// TIA Portal V17 program export: 3 tag tables, 4 data types, 12 data blocks, 34 code blocks (in call order from the OBs), 34 instance data blocks

VAR_GLOBAL   // PLC tag table "Input"
   I_D1 AT %I0.0 : Bool;
   I_D2 AT %I0.1 : Bool;
   I_D3 AT %I0.2 : Bool;
   I_D4 AT %I0.3 : Bool;
   I_D5 AT %I0.4 : Bool;
   I_D6 AT %I0.5 : Bool;
   I_D7 AT %I0.6 : Bool;
   I_D8 AT %I0.7 : Bool;
   I_D9 AT %I1.0 : Bool;
   I_Start AT %I1.1 : Bool;
   I_Reset AT %I1.2 : Bool;
   I_Stop AT %I1.3 : Bool;
   I_Auto AT %I1.4 : Bool;
   I_Manual AT %I1.5 : Bool;
   I_Estop AT %I1.6 : Bool;
   I_C1 AT %I1.7 : Bool;
   I_C2 AT %I2.0 : Bool;
   I_C3 AT %I2.1 : Bool;
   I_C4 AT %I2.2 : Bool;
   I_C5 AT %I2.3 : Bool;
   I_SendLeft AT %I2.4 : Bool;
   I_SendForward AT %I2.5 : Bool;
   I_SendRight AT %I2.6 : Bool;
   I_ResetCount AT %I2.7 : Bool;
   I_Weight AT %ID30 : Real;
END_VAR

VAR_GLOBAL   // PLC tag table "Output"
   O_W AT %Q0.0 : Bool;
   O_SendLeft AT %Q0.1 : Bool;
   O_SendRight AT %Q0.2 : Bool;
   O_SendForward AT %Q0.3 : Bool;
   O_StartLight AT %Q0.4 : Bool;
   O_ResetLight AT %Q0.5 : Bool;
   O_StopLight AT %Q0.6 : Bool;
   O_ColumnRed AT %Q0.7 : Bool;
   O_ColumnGreen AT %Q1.0 : Bool;
   O_ColumnYellow AT %Q1.1 : Bool;
   O_C1_light AT %Q1.2 : Bool;
   O_C3_light AT %Q1.4 : Bool;
   O_C4_light AT %Q1.5 : Bool;
   O_C5_light AT %Q1.6 : Bool;
   O_SendLeft_light AT %Q1.7 : Bool;
   O_SendForward_light AT %Q2.0 : Bool;
   O_SendRight_light AT %Q2.1 : Bool;
   O_ResetCount_light AT %Q2.2 : Bool;
   O_AlarmSiren AT %Q2.3 : Bool;
   O_C2_light AT %Q1.3 : Bool;
   O_LeftCount AT %QD30 : DInt;
   O_ForwardCount AT %QD34 : DInt;
   O_RightCOunt AT %QD38 : DInt;
   O_Weight AT %QD42 : Real;
   O_C1 AT %QD46 : DInt;
   O_C2 AT %QD50 : DInt;
   O_C3 AT %QD54 : DInt;
   O_C4 AT %QD58 : DInt;
END_VAR

VAR_GLOBAL   // PLC tag table "Standard-Variablentabelle"
   System_Byte AT %MB1 : Byte;
   FirstScan AT %M1.0 : Bool;
   DiagStatusUpdate AT %M1.1 : Bool;
   AlwaysTRUE AT %M1.2 : Bool;
   AlwaysFALSE AT %M1.3 : Bool;
   Clock_Byte AT %MB0 : Byte;
   Clock_10Hz AT %M0.0 : Bool;
   Clock_5Hz AT %M0.1 : Bool;
   "Clock_2.5Hz" AT %M0.2 : Bool;
   Clock_2Hz AT %M0.3 : Bool;
   "Clock_1.25Hz" AT %M0.4 : Bool;
   Clock_1Hz AT %M0.5 : Bool;
   "Clock_0.625Hz" AT %M0.6 : Bool;
   "Clock_0.5Hz" AT %M0.7 : Bool;
END_VAR

TYPE "stt_Conveyor"
// stored: IsFailsafeCompliant false
   STRUCT
      C1 : Bool;
      C2 { S7_SetPoint := 'True'} : Bool;
      C3 { S7_SetPoint := 'True'} : Bool;
      C4 { S7_SetPoint := 'True'} : Bool;
      W { S7_SetPoint := 'True'} : Bool;
      Left : Bool;
      Forward : Bool;
      Right : Bool;
   END_STRUCT;
END_TYPE

TYPE "stt_LostPackageError"
// stored: IsFailsafeCompliant false
   STRUCT
      Error_1 : Bool;
      Error_2 : Bool;
      Error_3 : Bool;
      Error_4 : Bool;
      Error_5 : Bool;
      Error_6 : Bool;
   END_STRUCT;
END_TYPE

TYPE "stt_Motor"
// stored: IsFailsafeCompliant false
   STRUCT
      Run : Bool;
      LeftTurn : Bool;
      RightTurn : Bool;
      Speed : Real;
   END_STRUCT;
END_TYPE

TYPE "stt_TimeWork"
// stored: IsFailsafeCompliant false
   STRUCT
      Seconds : USInt;
      Minute : USInt;
      Hours : USInt;
      Days : UDInt;
   END_STRUCT;
END_TYPE

DATA_BLOCK "ERR_ErrorData"   // DB27
{ S7_Optimized_Access := 'TRUE' }
VERSION : 0.1
// stored: AutoNumber true, IsOnlyStoredInLoadMemory false, IsRetainMemResEnabled false, IsWriteProtectedInAS false, MemoryReserve 100
   VAR
      ErrorChangeMode : Bool;
      ErrorEmergencyStop : Bool;
      ErrorLostPackage_B { S7_SetPoint := 'True'} : Bool;
      ErrorLostPackage : "stt_LostPackageError";
   END_VAR
BEGIN
END_DATA_BLOCK

DATA_BLOCK "TST_ChooseModeData"   // DB4
{ S7_Optimized_Access := 'TRUE' }
VERSION : 0.1
// stored: AutoNumber true, IsOnlyStoredInLoadMemory false, IsRetainMemResEnabled false, IsWriteProtectedInAS false, MemoryReserve 100
   VAR
      Auto : Bool;
      Manual : Bool;
      inAuto : Bool;
      inManual : Bool;
   END_VAR
BEGIN
END_DATA_BLOCK

DATA_BLOCK "TST_ControlLineData"   // DB7
{ S7_Optimized_Access := 'TRUE' }
VERSION : 0.1
// stored: AutoNumber true, IsOnlyStoredInLoadMemory false, IsRetainMemResEnabled false, IsWriteProtectedInAS false, MemoryReserve 100
   VAR
      inAuto : Bool;
      inManual : Bool;
      inStart : Bool;
      inStop : Bool;
      inGlobalError : Bool;
      inRunLine : Bool;
      StartLine : Bool;
      StopLine : Bool;
      StartAlarmSiren : Bool;
   END_VAR
BEGIN
END_DATA_BLOCK

DATA_BLOCK "LOG_LogicData"   // DB55
{ S7_Optimized_Access := 'TRUE' }
VERSION : 0.1
// stored: AutoNumber true, IsOnlyStoredInLoadMemory false, IsRetainMemResEnabled false, IsWriteProtectedInAS false, MemoryReserve 100
   VAR
      ConveyorsManual : "stt_Conveyor";
      ConveyorsAuto : "stt_Conveyor";
   END_VAR
BEGIN
END_DATA_BLOCK

DATA_BLOCK "HW_HardwareData"   // DB16
{ S7_Optimized_Access := 'TRUE' }
VERSION : 0.1
// stored: AutoNumber true, IsOnlyStoredInLoadMemory false, IsRetainMemResEnabled false, IsWriteProtectedInAS false, MemoryReserve 100
   VAR
      C1 : "stt_Motor";
      C2 { S7_SetPoint := 'True'} : "stt_Motor";
      C3 { S7_SetPoint := 'True'} : "stt_Motor";
      C4 { S7_SetPoint := 'True'} : "stt_Motor";
      W { S7_SetPoint := 'True'} : Bool;
      SendLeft : Bool;
      SendForward : Bool;
      SendRight : Bool;
   END_VAR
BEGIN
END_DATA_BLOCK

DATA_BLOCK "LOG_ConveyorWorkTime"   // DB47
{ S7_Optimized_Access := 'TRUE' }
VERSION : 0.1
// stored: AutoNumber true, IsOnlyStoredInLoadMemory false, IsRetainMemResEnabled false, IsWriteProtectedInAS false, MemoryReserve 20
   VAR RETAIN
      T1 { S7_SetPoint := 'True'} : "stt_TimeWork";
      T2 { S7_SetPoint := 'True'} : "stt_TimeWork";
      T3 { S7_SetPoint := 'True'} : "stt_TimeWork";
   END_VAR
   VAR
      T4 { S7_SetPoint := 'True'} : "stt_TimeWork";
      W { S7_SetPoint := 'True'} : "stt_TimeWork";
      O { S7_SetPoint := 'True'} : "stt_TimeWork";
   END_VAR
BEGIN
END_DATA_BLOCK

DATA_BLOCK "LOG_LineModeTurnOn"   // DB46
{ S7_Optimized_Access := 'TRUE' }
VERSION : 0.1
// stored: AutoNumber true, IsOnlyStoredInLoadMemory false, IsRetainMemResEnabled false, IsWriteProtectedInAS false, MemoryReserve 20
   VAR RETAIN
      ModeAuto : UDInt;
      ModeManual : UDInt;
   END_VAR
   VAR
      EmergencyButton : Int;
      ErrorLostPackage : UDInt;
      ErrorChangeMode : UDInt;
   END_VAR
BEGIN
END_DATA_BLOCK

DATA_BLOCK "LOG_LineTimeStatistic"   // DB44
{ S7_Optimized_Access := 'TRUE' }
VERSION : 0.1
// stored: AutoNumber true, IsOnlyStoredInLoadMemory false, IsRetainMemResEnabled false, IsWriteProtectedInAS false, MemoryReserve 20
   VAR RETAIN
      StartLine { S7_SetPoint := 'True'} : "stt_TimeWork";
      StopLine { S7_SetPoint := 'True'} : "stt_TimeWork";
      AutoMode { S7_SetPoint := 'True'} : "stt_TimeWork";
      ManualMode { S7_SetPoint := 'True'} : "stt_TimeWork";
      Error { S7_SetPoint := 'True'} : "stt_TimeWork";
   END_VAR
BEGIN
END_DATA_BLOCK

DATA_BLOCK "LOG_StatisticData"   // DB43
{ S7_Optimized_Access := 'TRUE' }
VERSION : 0.1
// stored: AutoNumber true, IsOnlyStoredInLoadMemory false, IsRetainMemResEnabled false, IsWriteProtectedInAS false, MemoryReserve 100
   VAR
      P_StartLine : Bool;
   END_VAR
BEGIN
END_DATA_BLOCK

DATA_BLOCK "LOG_TotalProduction"   // DB39
{ S7_Optimized_Access := 'TRUE' }
VERSION : 0.1
// stored: AutoNumber true, IsOnlyStoredInLoadMemory false, IsRetainMemResEnabled false, IsWriteProtectedInAS false, MemoryReserve 100
   VAR
      SmallPackage : Int;
      MediumPackage : Int;
      LargePackage : Int;
   END_VAR
BEGIN
END_DATA_BLOCK

DATA_BLOCK "HW_WeightData"   // DB22
{ S7_Optimized_Access := 'TRUE' }
VERSION : 0.1
// stored: AutoNumber true, IsOnlyStoredInLoadMemory false, IsRetainMemResEnabled false, IsWriteProtectedInAS false, MemoryReserve 100
   VAR
      WeightFilter : Real;
      P_D2 : Bool;
      WeightOfSmallPackage : Real;
      WeightOfLargePackage : Real;
      IsSmallPackage : Bool;
      IsMediumPackage : Bool;
      IsLargePackage : Bool;
   END_VAR
BEGIN
END_DATA_BLOCK

DATA_BLOCK "MAN_LineModeData"   // DB1
{ S7_Optimized_Access := 'TRUE' }
VERSION : 0.1
// stored: AutoNumber true, IsOnlyStoredInLoadMemory false, IsRetainMemResEnabled false, IsWriteProtectedInAS false, MemoryReserve 100
   VAR
      Start : Bool;
      Stop : Bool;
      Manual : Bool;
      Auto : Bool;
      Error : Bool;
      RunLine : Bool;
      AlarmSiren : Bool;
   END_VAR
BEGIN
END_DATA_BLOCK

ORGANIZATION_BLOCK "Main"   // OB1, LAD, ProgramCycle
TITLE = "Main Program Sweep (Cycle)"
{ S7_Optimized_Access := 'TRUE' }
VERSION : 0.1
// stored: AutoNumber true, IsIECCheckEnabled false, SetENOAutomatically false
   VAR_INPUT
      Initial_Call : Bool;   // Initial call of this OB
      Remanence : Bool;   // =True, if remanent data are available
   END_VAR
BEGIN

REGION Network 1: Connection of PLC with FactoryIO
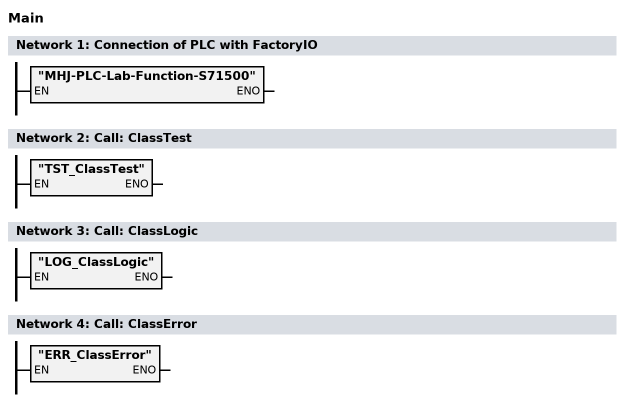
   RUNG wire#powerrail
      "MHJ-PLC-Lab-Function-S71500"()
   END_RUNG
   // the same network as SCL:
   "MHJ-PLC-Lab-Function-S71500"();
END_REGION

REGION Network 2: Call: ClassTest
   RUNG wire#powerrail
      "TST_ClassTest"()
   END_RUNG
   // the same network as SCL:
   "TST_ClassTest"();
END_REGION

REGION Network 3: Call: ClassLogic
   RUNG wire#powerrail
      "LOG_ClassLogic"()
   END_RUNG
   // the same network as SCL:
   "LOG_ClassLogic"();
END_REGION

REGION Network 4: Call: ClassError
   RUNG wire#powerrail
      "ERR_ClassError"()
   END_RUNG
   // the same network as SCL:
   "ERR_ClassError"();
END_REGION
END_ORGANIZATION_BLOCK

FUNCTION "TST_ClassTest" : Void   // FC2, LAD
{ S7_Optimized_Access := 'TRUE' }
VERSION : 0.1
// stored: AutoNumber true, IsIECCheckEnabled false, SetENOAutomatically false, UDAEnableTagReadback false
BEGIN

REGION Network 1: Call: ChooseMode
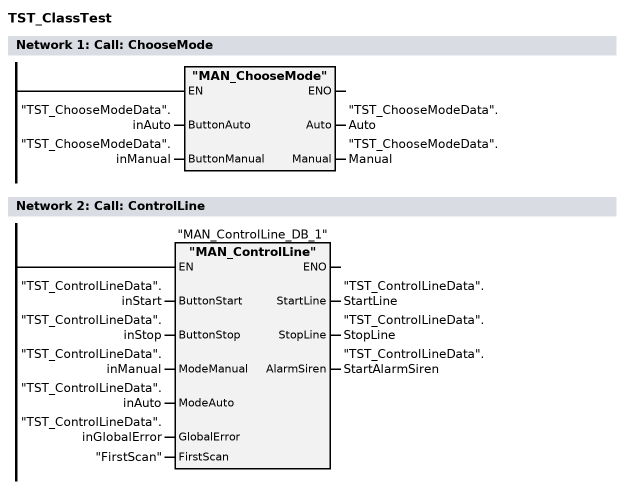
   RUNG wire#powerrail
      "MAN_ChooseMode"(ButtonAuto := "TST_ChooseModeData".inAuto, ButtonManual := "TST_ChooseModeData".inManual, Auto => "TST_ChooseModeData".Auto, Manual => "TST_ChooseModeData".Manual)
   END_RUNG
   // the same network as SCL:
   "MAN_ChooseMode"(ButtonAuto := "TST_ChooseModeData".inAuto,
                    ButtonManual := "TST_ChooseModeData".inManual,
                    Auto => "TST_ChooseModeData".Auto,
                    Manual => "TST_ChooseModeData".Manual);
END_REGION

REGION Network 2: Call: ControlLine
   RUNG wire#powerrail
      "MAN_ControlLine_DB_1"(ButtonStart := "TST_ControlLineData".inStart, ButtonStop := "TST_ControlLineData".inStop, ModeManual := "TST_ControlLineData".inManual, ModeAuto := "TST_ControlLineData".inAuto, GlobalError := "TST_ControlLineData".inGlobalError, FirstScan := "FirstScan", StartLine => "TST_ControlLineData".StartLine, StopLine => "TST_ControlLineData".StopLine, AlarmSiren => "TST_ControlLineData".StartAlarmSiren)
   END_RUNG
   // the same network as SCL:
   "MAN_ControlLine_DB_1"(ButtonStart := "TST_ControlLineData".inStart,   // "MAN_ControlLine"
                          ButtonStop := "TST_ControlLineData".inStop,
                          ModeManual := "TST_ControlLineData".inManual,
                          ModeAuto := "TST_ControlLineData".inAuto,
                          GlobalError := "TST_ControlLineData".inGlobalError,
                          FirstScan := "FirstScan",
                          StartLine => "TST_ControlLineData".StartLine,
                          StopLine => "TST_ControlLineData".StopLine,
                          AlarmSiren => "TST_ControlLineData".StartAlarmSiren);
END_REGION
END_FUNCTION

FUNCTION "MAN_ChooseMode" : Void   // FC7, LAD
{ S7_Optimized_Access := 'TRUE' }
VERSION : 0.1
// stored: AutoNumber true, IsIECCheckEnabled false, SetENOAutomatically false, UDAEnableTagReadback false
   VAR_INPUT
      ButtonAuto : Bool;
      ButtonManual : Bool;
   END_VAR
   VAR_OUTPUT
      Auto : Bool;
      Manual : Bool;
   END_VAR
BEGIN

REGION Network 1
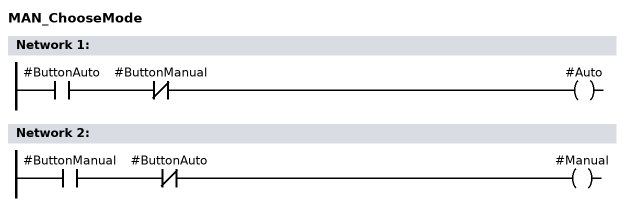
   RUNG wire#powerrail
      Contact( #ButtonAuto )
      I_Contact( #ButtonManual )
      Coil( #Auto )
   END_RUNG
   // the same network as SCL:
   #Auto := #ButtonAuto AND NOT #ButtonManual;
END_REGION

REGION Network 2
   RUNG wire#powerrail
      Contact( #ButtonManual )
      I_Contact( #ButtonAuto )
      Coil( #Manual )
   END_RUNG
   // the same network as SCL:
   #Manual := #ButtonManual AND NOT #ButtonAuto;
END_REGION
END_FUNCTION

FUNCTION_BLOCK "MAN_ControlLine"   // FB2, LAD
TITLE = Control Line - Sequential algorithm
{ S7_Optimized_Access := 'TRUE' }
VERSION : 0.1
// stored: AutoNumber true, IsIECCheckEnabled false, IsRetainMemResEnabled false, MemoryReserve 100, SetENOAutomatically false, UDAEnableTagReadback false
   VAR_INPUT
      ButtonStart : Bool;
      ButtonStop : Bool;
      ModeManual : Bool;
      ModeAuto : Bool;
      GlobalError : Bool;
      FirstScan : Bool;
   END_VAR
   VAR_OUTPUT
      StartLine : Bool;
      StopLine : Bool;
      AlarmSiren : Bool;
   END_VAR
   VAR
      s1 : Bool;
      s2 : Bool;
      s3 : Bool;
      s4 : Bool;
      P_ButtonStart_1 : Bool;
      P_ButtonStart_2 : Bool;
      IEC_Timer_0_Instance { ExternalAccessible := 'False'; ExternalVisible := 'False'; ExternalWritable := 'False'} : TP_TIME;
      Run { S7_SetPoint := 'True'} : Bool;
      N_Run : Bool;
   END_VAR
   VAR_TEMP   // added for the SCL form of the ladder/FBD networks
      _w1 : Bool;
   END_VAR
BEGIN

REGION Network 1: Step 2-1
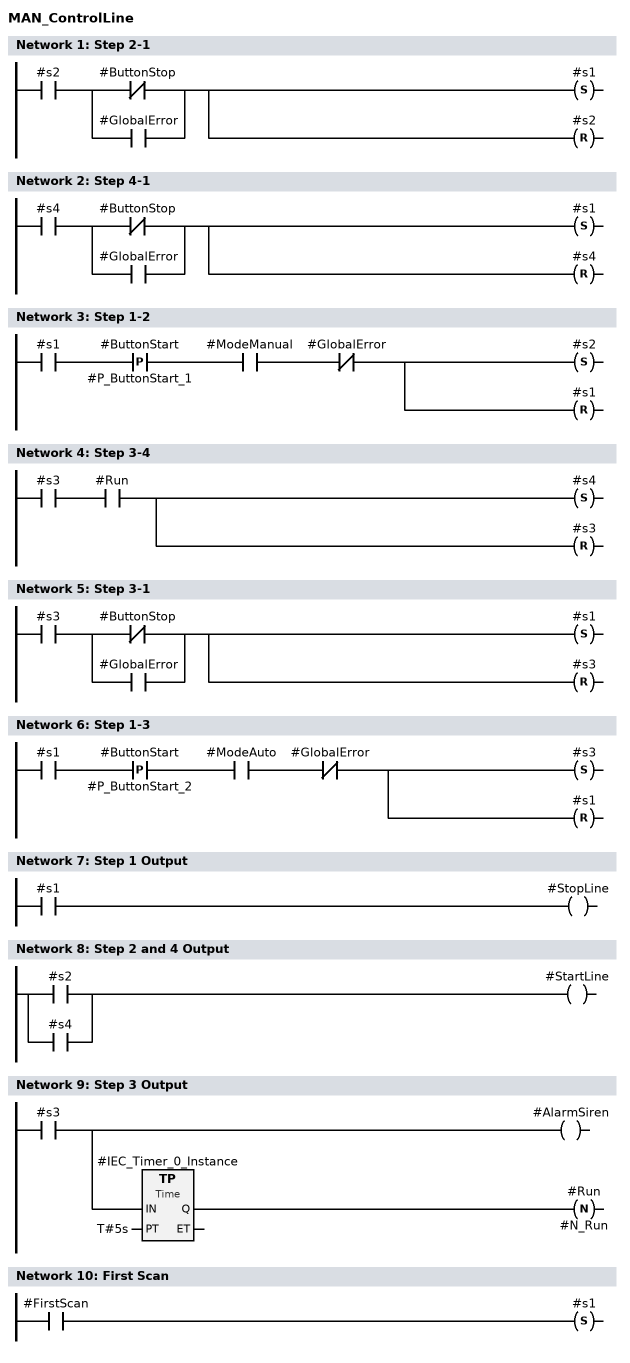
   RUNG wire#powerrail
      Contact( #s2 )
      wire#w1
      I_Contact( #ButtonStop )
      wire#w2
      S_Coil( #s1 )
   END_RUNG
   RUNG wire#w1
      Contact( #GlobalError )
   END_RUNG wire#w2
   RUNG wire#w2
      R_Coil( #s2 )
   END_RUNG
   // the same network as SCL:
   IF #s2 AND (NOT #ButtonStop OR #GlobalError) THEN
       #s1 := TRUE;
       #s2 := FALSE;
   END_IF;
END_REGION

REGION Network 2: Step 4-1
   RUNG wire#powerrail
      Contact( #s4 )
      wire#w1
      I_Contact( #ButtonStop )
      wire#w2
      S_Coil( #s1 )
   END_RUNG
   RUNG wire#w1
      Contact( #GlobalError )
   END_RUNG wire#w2
   RUNG wire#w2
      R_Coil( #s4 )
   END_RUNG
   // the same network as SCL:
   IF #s4 AND (NOT #ButtonStop OR #GlobalError) THEN
       #s1 := TRUE;
       #s4 := FALSE;
   END_IF;
END_REGION

REGION Network 3: Step 1-2
   RUNG wire#powerrail
      Contact( #s1 )
      P_Contact(operand := #ButtonStart, bit := #P_ButtonStart_1)
      Contact( #ModeManual )
      I_Contact( #GlobalError )
      wire#w1
      S_Coil( #s2 )
   END_RUNG
   RUNG wire#w1
      R_Coil( #s1 )
   END_RUNG
   // the same network as SCL:
   #_w1 := #s1 AND #ButtonStart AND NOT #P_ButtonStart_1;   // rising edge of #ButtonStart
   #P_ButtonStart_1 := #ButtonStart;
   IF #_w1 AND #ModeManual AND NOT #GlobalError THEN
       #s2 := TRUE;
       #s1 := FALSE;
   END_IF;
END_REGION

REGION Network 4: Step 3-4
   RUNG wire#powerrail
      Contact( #s3 )
      Contact( #Run )
      wire#w1
      S_Coil( #s4 )
   END_RUNG
   RUNG wire#w1
      R_Coil( #s3 )
   END_RUNG
   // the same network as SCL:
   IF #s3 AND #Run THEN
       #s4 := TRUE;
       #s3 := FALSE;
   END_IF;
END_REGION

REGION Network 5: Step 3-1
   RUNG wire#powerrail
      Contact( #s3 )
      wire#w1
      I_Contact( #ButtonStop )
      wire#w2
      S_Coil( #s1 )
   END_RUNG
   RUNG wire#w1
      Contact( #GlobalError )
   END_RUNG wire#w2
   RUNG wire#w2
      R_Coil( #s3 )
   END_RUNG
   // the same network as SCL:
   IF #s3 AND (NOT #ButtonStop OR #GlobalError) THEN
       #s1 := TRUE;
       #s3 := FALSE;
   END_IF;
END_REGION

REGION Network 6: Step 1-3
   RUNG wire#powerrail
      Contact( #s1 )
      P_Contact(operand := #ButtonStart, bit := #P_ButtonStart_2)
      Contact( #ModeAuto )
      I_Contact( #GlobalError )
      wire#w1
      S_Coil( #s3 )
   END_RUNG
   RUNG wire#w1
      R_Coil( #s1 )
   END_RUNG
   // the same network as SCL:
   #_w1 := #s1 AND #ButtonStart AND NOT #P_ButtonStart_2;   // rising edge of #ButtonStart
   #P_ButtonStart_2 := #ButtonStart;
   IF #_w1 AND #ModeAuto AND NOT #GlobalError THEN
       #s3 := TRUE;
       #s1 := FALSE;
   END_IF;
END_REGION

REGION Network 7: Step 1 Output
   RUNG wire#powerrail
      Contact( #s1 )
      Coil( #StopLine )
   END_RUNG
   // the same network as SCL:
   #StopLine := #s1;
END_REGION

REGION Network 8: Step 2 and 4 Output
   RUNG wire#powerrail
      Contact( #s2 )
      wire#w1
      Coil( #StartLine )
   END_RUNG
   RUNG wire#powerrail
      Contact( #s4 )
   END_RUNG wire#w1
   // the same network as SCL:
   #StartLine := #s2 OR #s4;
END_REGION

REGION Network 9: Step 3 Output
   #AlarmSiren := #s3;
   #IEC_Timer_0_Instance(IN := #s3, PT := T#5s);   // TP
   #Run := NOT #IEC_Timer_0_Instance.Q AND #N_Run;   // falling edge
   #N_Run := #IEC_Timer_0_Instance.Q;
END_REGION

REGION Network 10: First Scan
   RUNG wire#powerrail
      Contact( #FirstScan )
      S_Coil( #s1 )
   END_RUNG
   // the same network as SCL:
   IF #FirstScan THEN #s1 := TRUE; END_IF;
END_REGION
END_FUNCTION_BLOCK

FUNCTION "LOG_ClassLogic" : Void   // FC4, LAD
{ S7_Optimized_Access := 'TRUE' }
VERSION : 0.1
// stored: AutoNumber true, IsIECCheckEnabled false, SetENOAutomatically false, UDAEnableTagReadback false
BEGIN

REGION Network 1: Call: Mode
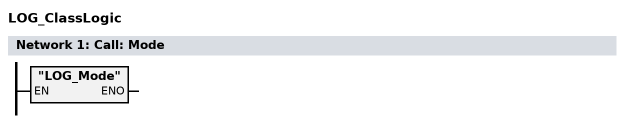
   RUNG wire#powerrail
      "LOG_Mode"()
   END_RUNG
   // the same network as SCL:
   "LOG_Mode"();
END_REGION
END_FUNCTION

FUNCTION "LOG_Mode" : Void   // FC13, LAD
{ S7_Optimized_Access := 'TRUE' }
VERSION : 0.1
// stored: AutoNumber true, IsIECCheckEnabled false, SetENOAutomatically false, UDAEnableTagReadback false
BEGIN

REGION Network 1: Call: AutoControle
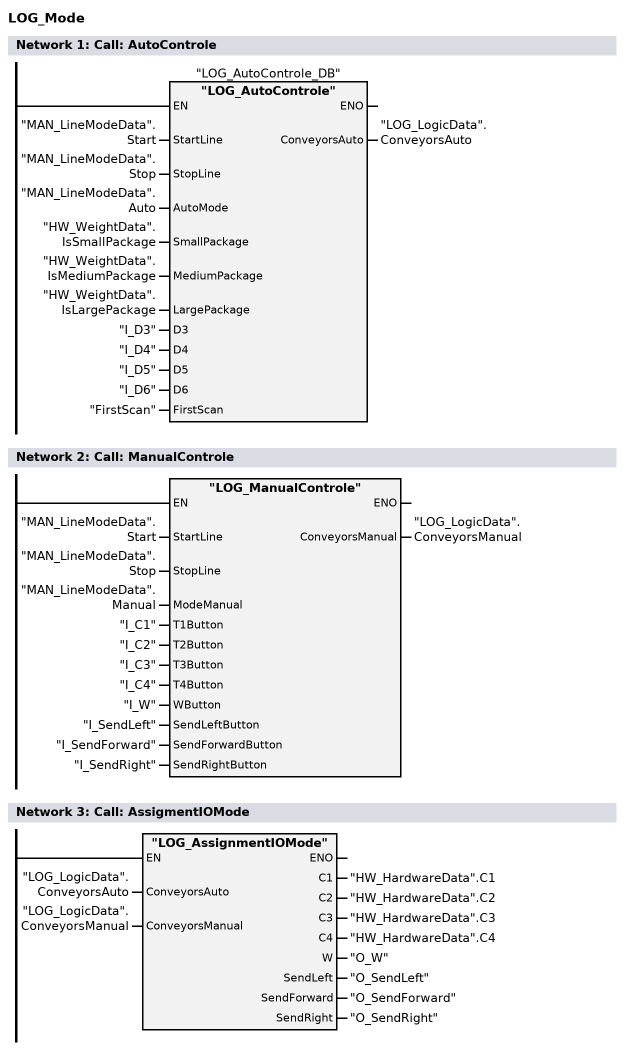
   RUNG wire#powerrail
      "LOG_AutoControle_DB"(StartLine := "MAN_LineModeData".Start, StopLine := "MAN_LineModeData".Stop, AutoMode := "MAN_LineModeData".Auto, SmallPackage := "HW_WeightData".IsSmallPackage, MediumPackage := "HW_WeightData".IsMediumPackage, LargePackage := "HW_WeightData".IsLargePackage, D3 := "I_D3", D4 := "I_D4", D5 := "I_D5", D6 := "I_D6", FirstScan := "FirstScan", ConveyorsAuto => "LOG_LogicData".ConveyorsAuto)
   END_RUNG
   // the same network as SCL:
   "LOG_AutoControle_DB"(StartLine := "MAN_LineModeData".Start,   // "LOG_AutoControle"
                         StopLine := "MAN_LineModeData".Stop,
                         AutoMode := "MAN_LineModeData".Auto,
                         SmallPackage := "HW_WeightData".IsSmallPackage,
                         MediumPackage := "HW_WeightData".IsMediumPackage,
                         LargePackage := "HW_WeightData".IsLargePackage,
                         D3 := "I_D3",
                         D4 := "I_D4",
                         D5 := "I_D5",
                         D6 := "I_D6",
                         FirstScan := "FirstScan",
                         ConveyorsAuto => "LOG_LogicData".ConveyorsAuto);
END_REGION

REGION Network 2: Call: ManualControle
   RUNG wire#powerrail
      "LOG_ManualControle"(StartLine := "MAN_LineModeData".Start, StopLine := "MAN_LineModeData".Stop, ModeManual := "MAN_LineModeData".Manual, T1Button := "I_C1", T2Button := "I_C2", T3Button := "I_C3", T4Button := "I_C4", WButton := "I_W", SendLeftButton := "I_SendLeft", SendForwardButton := "I_SendForward", SendRightButton := "I_SendRight", ConveyorsManual => "LOG_LogicData".ConveyorsManual)
   END_RUNG
   // the same network as SCL:
   "LOG_ManualControle"(StartLine := "MAN_LineModeData".Start,
                        StopLine := "MAN_LineModeData".Stop,
                        ModeManual := "MAN_LineModeData".Manual,
                        T1Button := "I_C1",
                        T2Button := "I_C2",
                        T3Button := "I_C3",
                        T4Button := "I_C4",
                        WButton := "I_W",
                        SendLeftButton := "I_SendLeft",
                        SendForwardButton := "I_SendForward",
                        SendRightButton := "I_SendRight",
                        ConveyorsManual => "LOG_LogicData".ConveyorsManual);
END_REGION

REGION Network 3: Call: AssigmentIOMode
   RUNG wire#powerrail
      "LOG_AssignmentIOMode"(ConveyorsAuto := "LOG_LogicData".ConveyorsAuto, ConveyorsManual := "LOG_LogicData".ConveyorsManual, C1 => "HW_HardwareData".C1, C2 => "HW_HardwareData".C2, C3 => "HW_HardwareData".C3, C4 => "HW_HardwareData".C4, W => "O_W", SendLeft => "O_SendLeft", SendForward => "O_SendForward", SendRight => "O_SendRight")
   END_RUNG
   // the same network as SCL:
   "LOG_AssignmentIOMode"(ConveyorsAuto := "LOG_LogicData".ConveyorsAuto,
                          ConveyorsManual := "LOG_LogicData".ConveyorsManual,
                          C1 => "HW_HardwareData".C1,
                          C2 => "HW_HardwareData".C2,
                          C3 => "HW_HardwareData".C3,
                          C4 => "HW_HardwareData".C4,
                          W => "O_W",
                          SendLeft => "O_SendLeft",
                          SendForward => "O_SendForward",
                          SendRight => "O_SendRight");
END_REGION
END_FUNCTION

FUNCTION_BLOCK "LOG_AutoControle"   // FB5, LAD
TITLE = Auto Controle - Sequential algorithm
{ S7_Optimized_Access := 'TRUE' }
VERSION : 0.1
// stored: AutoNumber true, IsIECCheckEnabled false, IsRetainMemResEnabled false, MemoryReserve 100, SetENOAutomatically false, UDAEnableTagReadback false
   VAR_INPUT
      StartLine : Bool;
      StopLine : Bool;
      AutoMode : Bool;
      SmallPackage : Bool;
      MediumPackage : Bool;
      LargePackage : Bool;
      D3 : Bool;
      D4 : Bool;
      D5 : Bool;
      D6 : Bool;
      FirstScan : Bool;
   END_VAR
   VAR_OUTPUT
      ConveyorsAuto : "stt_Conveyor";
   END_VAR
   VAR
      s1 : Bool;
      s2 : Bool;
      s3 : Bool;
      s4 : Bool;
      s5 : Bool;
      P_D3_1 : Bool;
      P_D3_2 : Bool;
      P_D3_3 : Bool;
      N_D4 : Bool;
      N_D5 : Bool;
      N_D6 : Bool;
   END_VAR
   VAR_TEMP   // added for the SCL form of the ladder/FBD networks
      _w1 : Bool;
   END_VAR
BEGIN

REGION Network 1: Step 3-2
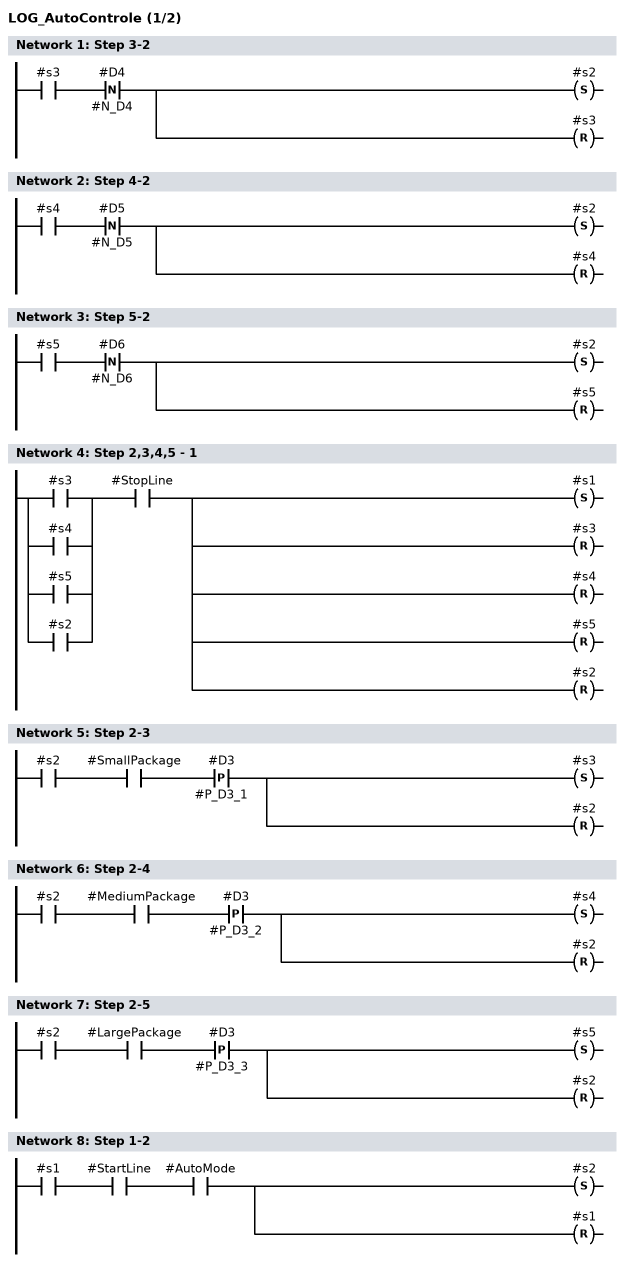
   RUNG wire#powerrail
      Contact( #s3 )
      N_Contact(operand := #D4, bit := #N_D4)
      wire#w1
      S_Coil( #s2 )
   END_RUNG
   RUNG wire#w1
      R_Coil( #s3 )
   END_RUNG
   // the same network as SCL:
   #_w1 := #s3 AND NOT #D4 AND #N_D4;   // falling edge of #D4
   #N_D4 := #D4;
   IF #_w1 THEN
       #s2 := TRUE;
       #s3 := FALSE;
   END_IF;
END_REGION

REGION Network 2: Step 4-2
   RUNG wire#powerrail
      Contact( #s4 )
      N_Contact(operand := #D5, bit := #N_D5)
      wire#w1
      S_Coil( #s2 )
   END_RUNG
   RUNG wire#w1
      R_Coil( #s4 )
   END_RUNG
   // the same network as SCL:
   #_w1 := #s4 AND NOT #D5 AND #N_D5;   // falling edge of #D5
   #N_D5 := #D5;
   IF #_w1 THEN
       #s2 := TRUE;
       #s4 := FALSE;
   END_IF;
END_REGION

REGION Network 3: Step 5-2
   RUNG wire#powerrail
      Contact( #s5 )
      N_Contact(operand := #D6, bit := #N_D6)
      wire#w1
      S_Coil( #s2 )
   END_RUNG
   RUNG wire#w1
      R_Coil( #s5 )
   END_RUNG
   // the same network as SCL:
   #_w1 := #s5 AND NOT #D6 AND #N_D6;   // falling edge of #D6
   #N_D6 := #D6;
   IF #_w1 THEN
       #s2 := TRUE;
       #s5 := FALSE;
   END_IF;
END_REGION

REGION Network 4: Step 2,3,4,5 - 1
   RUNG wire#powerrail
      Contact( #s3 )
      wire#w1
      Contact( #StopLine )
      wire#w2
      S_Coil( #s1 )
   END_RUNG
   RUNG wire#powerrail
      Contact( #s4 )
   END_RUNG wire#w1
   RUNG wire#powerrail
      Contact( #s5 )
   END_RUNG wire#w1
   RUNG wire#powerrail
      Contact( #s2 )
   END_RUNG wire#w1
   RUNG wire#w2
      R_Coil( #s3 )
   END_RUNG
   RUNG wire#w2
      R_Coil( #s4 )
   END_RUNG
   RUNG wire#w2
      R_Coil( #s5 )
   END_RUNG
   RUNG wire#w2
      R_Coil( #s2 )
   END_RUNG
   // the same network as SCL:
   IF (#s3 OR #s4 OR #s5 OR #s2) AND #StopLine THEN #s1 := TRUE; END_IF;
   #_w1 := (#s3 OR #s4 OR #s5 OR #s2) AND #StopLine;
   IF #_w1 THEN
       #s3 := FALSE;
       #s4 := FALSE;
       #s5 := FALSE;
       #s2 := FALSE;
   END_IF;
END_REGION

REGION Network 5: Step 2-3
   RUNG wire#powerrail
      Contact( #s2 )
      Contact( #SmallPackage )
      P_Contact(operand := #D3, bit := #P_D3_1)
      wire#w1
      S_Coil( #s3 )
   END_RUNG
   RUNG wire#w1
      R_Coil( #s2 )
   END_RUNG
   // the same network as SCL:
   #_w1 := #s2 AND #SmallPackage AND #D3 AND NOT #P_D3_1;   // rising edge of #D3
   #P_D3_1 := #D3;
   IF #_w1 THEN
       #s3 := TRUE;
       #s2 := FALSE;
   END_IF;
END_REGION

REGION Network 6: Step 2-4
   RUNG wire#powerrail
      Contact( #s2 )
      Contact( #MediumPackage )
      P_Contact(operand := #D3, bit := #P_D3_2)
      wire#w1
      S_Coil( #s4 )
   END_RUNG
   RUNG wire#w1
      R_Coil( #s2 )
   END_RUNG
   // the same network as SCL:
   #_w1 := #s2 AND #MediumPackage AND #D3 AND NOT #P_D3_2;   // rising edge of #D3
   #P_D3_2 := #D3;
   IF #_w1 THEN
       #s4 := TRUE;
       #s2 := FALSE;
   END_IF;
END_REGION

REGION Network 7: Step 2-5
   RUNG wire#powerrail
      Contact( #s2 )
      Contact( #LargePackage )
      P_Contact(operand := #D3, bit := #P_D3_3)
      wire#w1
      S_Coil( #s5 )
   END_RUNG
   RUNG wire#w1
      R_Coil( #s2 )
   END_RUNG
   // the same network as SCL:
   #_w1 := #s2 AND #LargePackage AND #D3 AND NOT #P_D3_3;   // rising edge of #D3
   #P_D3_3 := #D3;
   IF #_w1 THEN
       #s5 := TRUE;
       #s2 := FALSE;
   END_IF;
END_REGION

REGION Network 8: Step 1-2
   RUNG wire#powerrail
      Contact( #s1 )
      Contact( #StartLine )
      Contact( #AutoMode )
      wire#w1
      S_Coil( #s2 )
   END_RUNG
   RUNG wire#w1
      R_Coil( #s1 )
   END_RUNG
   // the same network as SCL:
   IF #s1 AND #StartLine AND #AutoMode THEN
       #s2 := TRUE;
       #s1 := FALSE;
   END_IF;
END_REGION

REGION Network 9: Step 2,3,4,5 Output
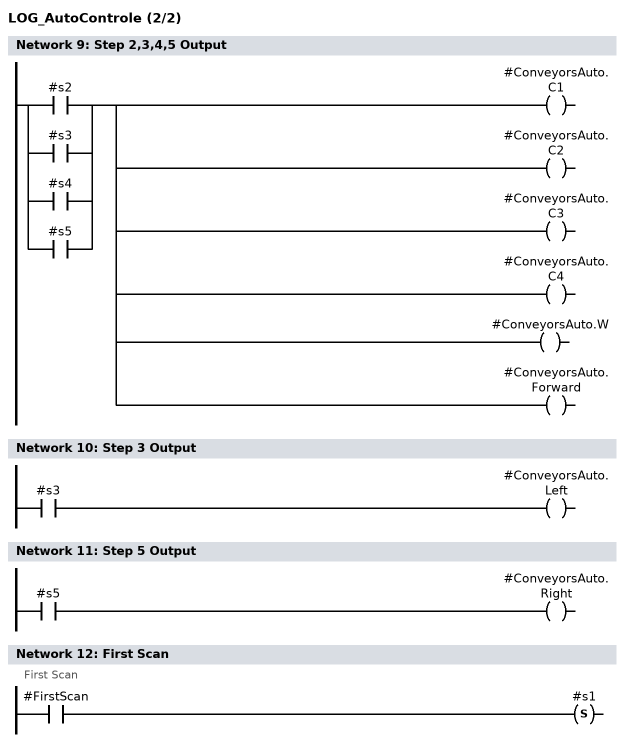
   RUNG wire#powerrail
      Contact( #s2 )
      wire#w1
      Coil( #ConveyorsAuto.C1 )
   END_RUNG
   RUNG wire#powerrail
      Contact( #s3 )
   END_RUNG wire#w1
   RUNG wire#powerrail
      Contact( #s4 )
   END_RUNG wire#w1
   RUNG wire#powerrail
      Contact( #s5 )
   END_RUNG wire#w1
   RUNG wire#w1
      Coil( #ConveyorsAuto.C2 )
   END_RUNG
   RUNG wire#w1
      Coil( #ConveyorsAuto.C3 )
   END_RUNG
   RUNG wire#w1
      Coil( #ConveyorsAuto.C4 )
   END_RUNG
   RUNG wire#w1
      Coil( #ConveyorsAuto.W )
   END_RUNG
   RUNG wire#w1
      Coil( #ConveyorsAuto.Forward )
   END_RUNG
   // the same network as SCL:
   #ConveyorsAuto.C1 := #s2 OR #s3 OR #s4 OR #s5;
   #ConveyorsAuto.C2 := #ConveyorsAuto.C1;
   #ConveyorsAuto.C3 := #ConveyorsAuto.C1;
   #ConveyorsAuto.C4 := #ConveyorsAuto.C1;
   #ConveyorsAuto.W := #ConveyorsAuto.C1;
   #ConveyorsAuto.Forward := #ConveyorsAuto.C1;
END_REGION

REGION Network 10: Step 3 Output
   RUNG wire#powerrail
      Contact( #s3 )
      Coil( #ConveyorsAuto.Left )
   END_RUNG
   // the same network as SCL:
   #ConveyorsAuto.Left := #s3;
END_REGION

REGION Network 11: Step 5 Output
   RUNG wire#powerrail
      Contact( #s5 )
      Coil( #ConveyorsAuto.Right )
   END_RUNG
   // the same network as SCL:
   #ConveyorsAuto.Right := #s5;
END_REGION

REGION Network 12: First Scan
   // First Scan
   RUNG wire#powerrail
      Contact( #FirstScan )
      S_Coil( #s1 )
   END_RUNG
   // the same network as SCL:
   IF #FirstScan THEN #s1 := TRUE; END_IF;
END_REGION
END_FUNCTION_BLOCK

FUNCTION "LOG_ManualControle" : Void   // FC10, LAD
{ S7_Optimized_Access := 'TRUE' }
VERSION : 0.1
// stored: AutoNumber true, IsIECCheckEnabled false, SetENOAutomatically false, UDAEnableTagReadback false
   VAR_INPUT
      StartLine : Bool;
      StopLine : Bool;
      ModeManual : Bool;
      T1Button : Bool;
      T2Button : Bool;
      T3Button : Bool;
      T4Button : Bool;
      WButton : Bool;
      SendLeftButton : Bool;
      SendForwardButton : Bool;
      SendRightButton : Bool;
   END_VAR
   VAR_OUTPUT
      ConveyorsManual : "stt_Conveyor";
   END_VAR
BEGIN

REGION Network 1: Call: ManualModule - C1
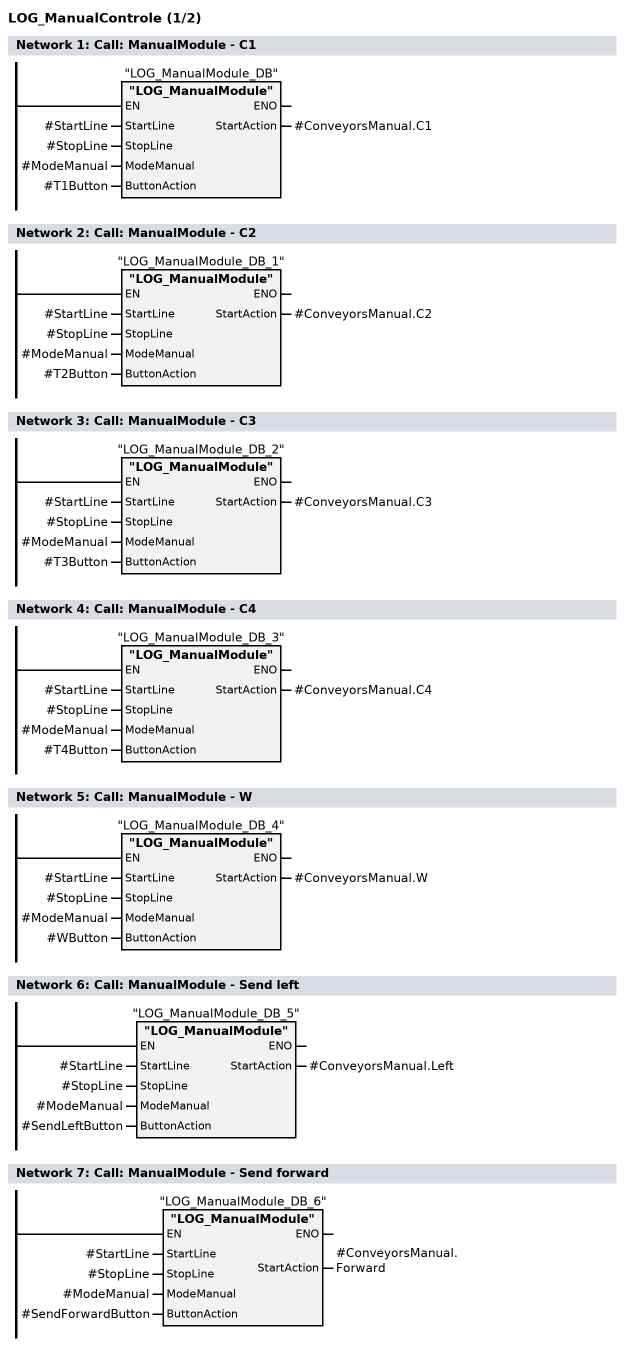
   RUNG wire#powerrail
      "LOG_ManualModule_DB"(StartLine := #StartLine, StopLine := #StopLine, ModeManual := #ModeManual, ButtonAction := #T1Button, StartAction => #ConveyorsManual.C1)
   END_RUNG
   // the same network as SCL:
   "LOG_ManualModule_DB"(StartLine := #StartLine,   // "LOG_ManualModule"
                         StopLine := #StopLine,
                         ModeManual := #ModeManual,
                         ButtonAction := #T1Button,
                         StartAction => #ConveyorsManual.C1);
END_REGION

REGION Network 2: Call: ManualModule - C2
   RUNG wire#powerrail
      "LOG_ManualModule_DB_1"(StartLine := #StartLine, StopLine := #StopLine, ModeManual := #ModeManual, ButtonAction := #T2Button, StartAction => #ConveyorsManual.C2)
   END_RUNG
   // the same network as SCL:
   "LOG_ManualModule_DB_1"(StartLine := #StartLine,   // "LOG_ManualModule"
                           StopLine := #StopLine,
                           ModeManual := #ModeManual,
                           ButtonAction := #T2Button,
                           StartAction => #ConveyorsManual.C2);
END_REGION

REGION Network 3: Call: ManualModule - C3
   RUNG wire#powerrail
      "LOG_ManualModule_DB_2"(StartLine := #StartLine, StopLine := #StopLine, ModeManual := #ModeManual, ButtonAction := #T3Button, StartAction => #ConveyorsManual.C3)
   END_RUNG
   // the same network as SCL:
   "LOG_ManualModule_DB_2"(StartLine := #StartLine,   // "LOG_ManualModule"
                           StopLine := #StopLine,
                           ModeManual := #ModeManual,
                           ButtonAction := #T3Button,
                           StartAction => #ConveyorsManual.C3);
END_REGION

REGION Network 4: Call: ManualModule - C4
   RUNG wire#powerrail
      "LOG_ManualModule_DB_3"(StartLine := #StartLine, StopLine := #StopLine, ModeManual := #ModeManual, ButtonAction := #T4Button, StartAction => #ConveyorsManual.C4)
   END_RUNG
   // the same network as SCL:
   "LOG_ManualModule_DB_3"(StartLine := #StartLine,   // "LOG_ManualModule"
                           StopLine := #StopLine,
                           ModeManual := #ModeManual,
                           ButtonAction := #T4Button,
                           StartAction => #ConveyorsManual.C4);
END_REGION

REGION Network 5: Call: ManualModule - W
   RUNG wire#powerrail
      "LOG_ManualModule_DB_4"(StartLine := #StartLine, StopLine := #StopLine, ModeManual := #ModeManual, ButtonAction := #WButton, StartAction => #ConveyorsManual.W)
   END_RUNG
   // the same network as SCL:
   "LOG_ManualModule_DB_4"(StartLine := #StartLine,   // "LOG_ManualModule"
                           StopLine := #StopLine,
                           ModeManual := #ModeManual,
                           ButtonAction := #WButton,
                           StartAction => #ConveyorsManual.W);
END_REGION

REGION Network 6: Call: ManualModule - Send left
   RUNG wire#powerrail
      "LOG_ManualModule_DB_5"(StartLine := #StartLine, StopLine := #StopLine, ModeManual := #ModeManual, ButtonAction := #SendLeftButton, StartAction => #ConveyorsManual.Left)
   END_RUNG
   // the same network as SCL:
   "LOG_ManualModule_DB_5"(StartLine := #StartLine,   // "LOG_ManualModule"
                           StopLine := #StopLine,
                           ModeManual := #ModeManual,
                           ButtonAction := #SendLeftButton,
                           StartAction => #ConveyorsManual.Left);
END_REGION

REGION Network 7: Call: ManualModule - Send forward
   RUNG wire#powerrail
      "LOG_ManualModule_DB_6"(StartLine := #StartLine, StopLine := #StopLine, ModeManual := #ModeManual, ButtonAction := #SendForwardButton, StartAction => #ConveyorsManual.Forward)
   END_RUNG
   // the same network as SCL:
   "LOG_ManualModule_DB_6"(StartLine := #StartLine,   // "LOG_ManualModule"
                           StopLine := #StopLine,
                           ModeManual := #ModeManual,
                           ButtonAction := #SendForwardButton,
                           StartAction => #ConveyorsManual.Forward);
END_REGION

REGION Network 8: Call: ManualModule - Send right
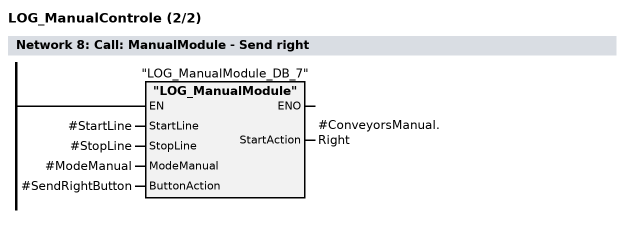
   RUNG wire#powerrail
      "LOG_ManualModule_DB_7"(StartLine := #StartLine, StopLine := #StopLine, ModeManual := #ModeManual, ButtonAction := #SendRightButton, StartAction => #ConveyorsManual.Right)
   END_RUNG
   // the same network as SCL:
   "LOG_ManualModule_DB_7"(StartLine := #StartLine,   // "LOG_ManualModule"
                           StopLine := #StopLine,
                           ModeManual := #ModeManual,
                           ButtonAction := #SendRightButton,
                           StartAction => #ConveyorsManual.Right);
END_REGION
END_FUNCTION

FUNCTION_BLOCK "LOG_ManualModule"   // FB14, LAD
{ S7_Optimized_Access := 'TRUE' }
VERSION : 0.1
// stored: AutoNumber true, IsIECCheckEnabled false, IsRetainMemResEnabled false, MemoryReserve 100, SetENOAutomatically false, UDAEnableTagReadback false
   VAR_INPUT
      StartLine : Bool;
      StopLine : Bool;
      ModeManual : Bool;
      ButtonAction : Bool;
   END_VAR
   VAR_OUTPUT
      StartAction : Bool;
   END_VAR
   VAR RETAIN
      IEC_Counter_0_Instance { ExternalAccessible := 'False'; ExternalVisible := 'False'; ExternalWritable := 'False'} : CTU_INT;
   END_VAR
   VAR
      P_ButtonAction : Bool;
      CV : Int;
      Reset : Bool;
   END_VAR
   VAR_TEMP   // added for the SCL form of the ladder/FBD networks
      _w1 : Bool;
   END_VAR
BEGIN

REGION Network 1
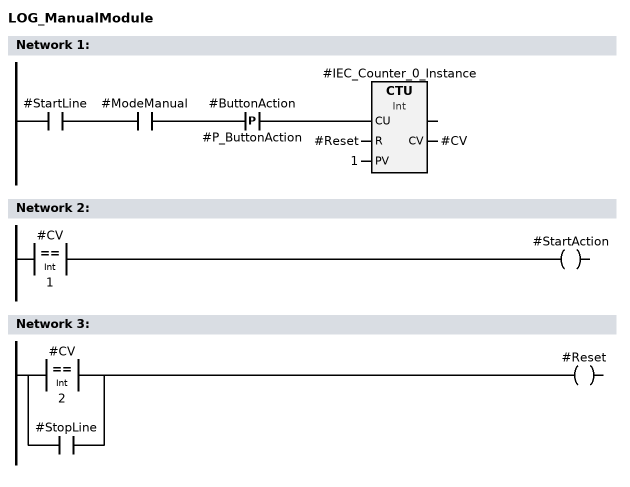
   RUNG wire#powerrail
      Contact( #StartLine )
      Contact( #ModeManual )
      P_Contact(operand := #ButtonAction, bit := #P_ButtonAction)
      { S7_Templates := "value_type := Int" } #IEC_Counter_0_Instance.CTU(r := #Reset, pv := 1, cv => #CV)
   END_RUNG
   // the same network as SCL:
   #_w1 := #StartLine AND #ModeManual AND #ButtonAction AND NOT #P_ButtonAction;   // rising edge of #ButtonAction
   #P_ButtonAction := #ButtonAction;
   #IEC_Counter_0_Instance(CU := #_w1, R := #Reset, PV := 1, CV => #CV);   // CTU
END_REGION

REGION Network 2
   RUNG wire#powerrail
      { S7_Templates := "SrcType := Int" } EQ_Contact(in1 := #CV, in2 := 1)
      Coil( #StartAction )
   END_RUNG
   // the same network as SCL:
   #StartAction := #CV = 1;
END_REGION

REGION Network 3
   RUNG wire#powerrail
      { S7_Templates := "SrcType := Int" } EQ_Contact(in1 := #CV, in2 := 2)
      wire#w1
      Coil( #Reset )
   END_RUNG
   RUNG wire#powerrail
      Contact( #StopLine )
   END_RUNG wire#w1
   // the same network as SCL:
   #Reset := (#CV = 2) OR #StopLine;
END_REGION
END_FUNCTION_BLOCK

FUNCTION "LOG_AssignmentIOMode" : Void   // FC26, LAD
{ S7_Optimized_Access := 'TRUE' }
VERSION : 0.1
// stored: AutoNumber true, IsIECCheckEnabled false, SetENOAutomatically false, UDAEnableTagReadback false
   VAR_INPUT
      ConveyorsAuto : "stt_Conveyor";
      ConveyorsManual : "stt_Conveyor";
   END_VAR
   VAR_OUTPUT
      C1 : "stt_Motor";
      C2 : "stt_Motor";
      C3 : "stt_Motor";
      C4 : "stt_Motor";
      W : Bool;
      SendLeft : Bool;
      SendForward : Bool;
      SendRight : Bool;
   END_VAR
BEGIN

REGION Network 1: C1
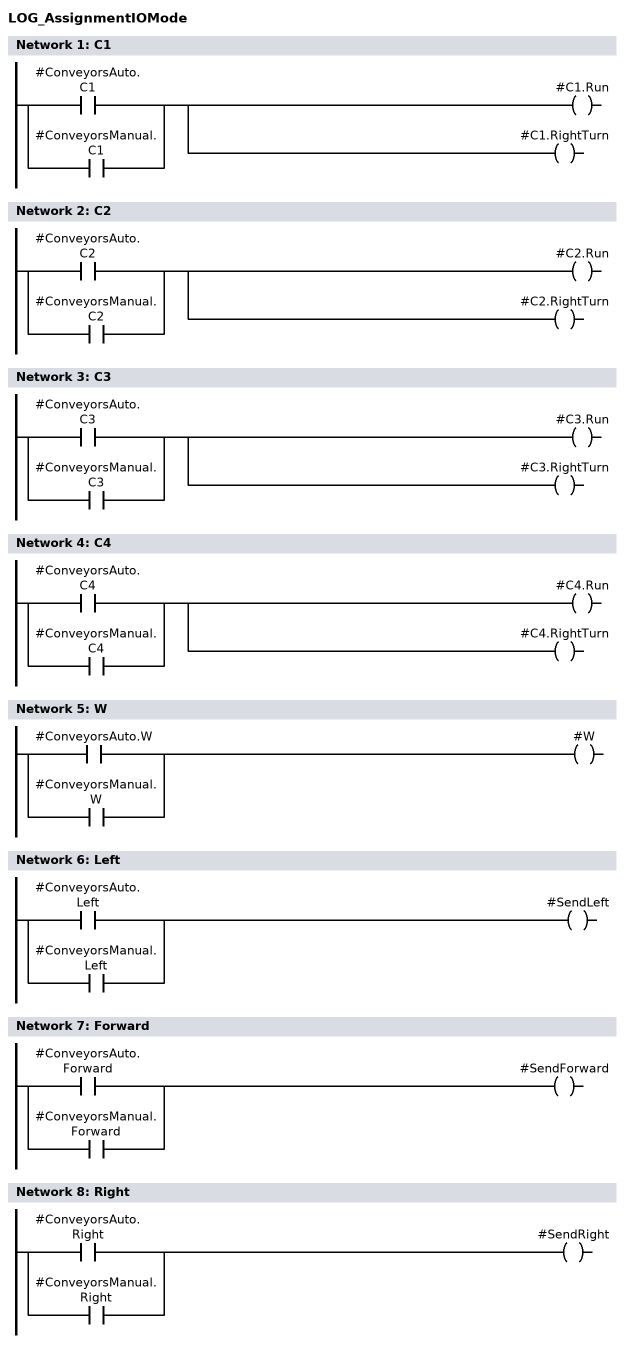
   RUNG wire#powerrail
      Contact( #ConveyorsAuto.C1 )
      wire#w1
      Coil( #C1.Run )
   END_RUNG
   RUNG wire#powerrail
      Contact( #ConveyorsManual.C1 )
   END_RUNG wire#w1
   RUNG wire#w1
      Coil( #C1.RightTurn )
   END_RUNG
   // the same network as SCL:
   #C1.Run := #ConveyorsAuto.C1 OR #ConveyorsManual.C1;
   #C1.RightTurn := #C1.Run;
END_REGION

REGION Network 2: C2
   RUNG wire#powerrail
      Contact( #ConveyorsAuto.C2 )
      wire#w1
      Coil( #C2.Run )
   END_RUNG
   RUNG wire#powerrail
      Contact( #ConveyorsManual.C2 )
   END_RUNG wire#w1
   RUNG wire#w1
      Coil( #C2.RightTurn )
   END_RUNG
   // the same network as SCL:
   #C2.Run := #ConveyorsAuto.C2 OR #ConveyorsManual.C2;
   #C2.RightTurn := #C2.Run;
END_REGION

REGION Network 3: C3
   RUNG wire#powerrail
      Contact( #ConveyorsAuto.C3 )
      wire#w1
      Coil( #C3.Run )
   END_RUNG
   RUNG wire#powerrail
      Contact( #ConveyorsManual.C3 )
   END_RUNG wire#w1
   RUNG wire#w1
      Coil( #C3.RightTurn )
   END_RUNG
   // the same network as SCL:
   #C3.Run := #ConveyorsAuto.C3 OR #ConveyorsManual.C3;
   #C3.RightTurn := #C3.Run;
END_REGION

REGION Network 4: C4
   RUNG wire#powerrail
      Contact( #ConveyorsAuto.C4 )
      wire#w1
      Coil( #C4.Run )
   END_RUNG
   RUNG wire#powerrail
      Contact( #ConveyorsManual.C4 )
   END_RUNG wire#w1
   RUNG wire#w1
      Coil( #C4.RightTurn )
   END_RUNG
   // the same network as SCL:
   #C4.Run := #ConveyorsAuto.C4 OR #ConveyorsManual.C4;
   #C4.RightTurn := #C4.Run;
END_REGION

REGION Network 5: W
   RUNG wire#powerrail
      Contact( #ConveyorsAuto.W )
      wire#w1
      Coil( #W )
   END_RUNG
   RUNG wire#powerrail
      Contact( #ConveyorsManual.W )
   END_RUNG wire#w1
   // the same network as SCL:
   #W := #ConveyorsAuto.W OR #ConveyorsManual.W;
END_REGION

REGION Network 6: Left
   RUNG wire#powerrail
      Contact( #ConveyorsAuto.Left )
      wire#w1
      Coil( #SendLeft )
   END_RUNG
   RUNG wire#powerrail
      Contact( #ConveyorsManual.Left )
   END_RUNG wire#w1
   // the same network as SCL:
   #SendLeft := #ConveyorsAuto.Left OR #ConveyorsManual.Left;
END_REGION

REGION Network 7: Forward
   RUNG wire#powerrail
      Contact( #ConveyorsAuto.Forward )
      wire#w1
      Coil( #SendForward )
   END_RUNG
   RUNG wire#powerrail
      Contact( #ConveyorsManual.Forward )
   END_RUNG wire#w1
   // the same network as SCL:
   #SendForward := #ConveyorsAuto.Forward OR #ConveyorsManual.Forward;
END_REGION

REGION Network 8: Right
   RUNG wire#powerrail
      Contact( #ConveyorsAuto.Right )
      wire#w1
      Coil( #SendRight )
   END_RUNG
   RUNG wire#powerrail
      Contact( #ConveyorsManual.Right )
   END_RUNG wire#w1
   // the same network as SCL:
   #SendRight := #ConveyorsAuto.Right OR #ConveyorsManual.Right;
END_REGION
END_FUNCTION

FUNCTION "ERR_ClassError" : Void   // FC1, LAD
{ S7_Optimized_Access := 'TRUE' }
VERSION : 0.1
// stored: AutoNumber true, IsIECCheckEnabled false, SetENOAutomatically false, UDAEnableTagReadback false
BEGIN

REGION Network 1: Call: EStop
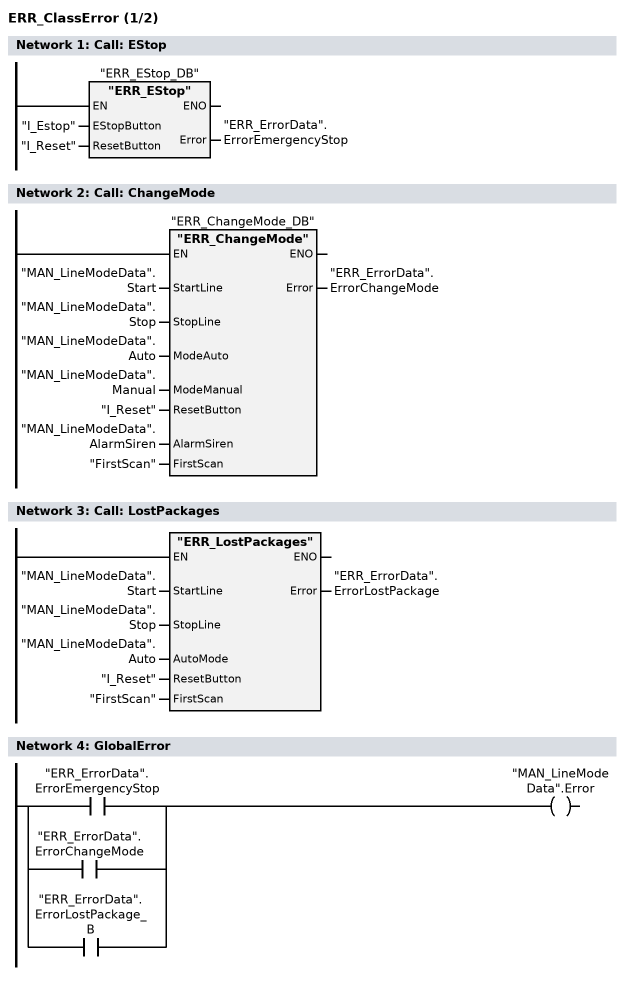
   RUNG wire#powerrail
      "ERR_EStop_DB"(EStopButton := "I_Estop", ResetButton := "I_Reset", Error => "ERR_ErrorData".ErrorEmergencyStop)
   END_RUNG
   // the same network as SCL:
   "ERR_EStop_DB"(EStopButton := "I_Estop",   // "ERR_EStop"
                  ResetButton := "I_Reset",
                  Error => "ERR_ErrorData".ErrorEmergencyStop);
END_REGION

REGION Network 2: Call: ChangeMode
   RUNG wire#powerrail
      "ERR_ChangeMode_DB"(StartLine := "MAN_LineModeData".Start, StopLine := "MAN_LineModeData".Stop, ModeAuto := "MAN_LineModeData".Auto, ModeManual := "MAN_LineModeData".Manual, ResetButton := "I_Reset", AlarmSiren := "MAN_LineModeData".AlarmSiren, FirstScan := "FirstScan", Error => "ERR_ErrorData".ErrorChangeMode)
   END_RUNG
   // the same network as SCL:
   "ERR_ChangeMode_DB"(StartLine := "MAN_LineModeData".Start,   // "ERR_ChangeMode"
                       StopLine := "MAN_LineModeData".Stop,
                       ModeAuto := "MAN_LineModeData".Auto,
                       ModeManual := "MAN_LineModeData".Manual,
                       ResetButton := "I_Reset",
                       AlarmSiren := "MAN_LineModeData".AlarmSiren,
                       FirstScan := "FirstScan",
                       Error => "ERR_ErrorData".ErrorChangeMode);
END_REGION

REGION Network 3: Call: LostPackages
   RUNG wire#powerrail
      "ERR_LostPackages"(StartLine := "MAN_LineModeData".Start, StopLine := "MAN_LineModeData".Stop, AutoMode := "MAN_LineModeData".Auto, ResetButton := "I_Reset", FirstScan := "FirstScan", Error => "ERR_ErrorData".ErrorLostPackage)
   END_RUNG
   // the same network as SCL:
   "ERR_LostPackages"(StartLine := "MAN_LineModeData".Start,
                      StopLine := "MAN_LineModeData".Stop,
                      AutoMode := "MAN_LineModeData".Auto,
                      ResetButton := "I_Reset",
                      FirstScan := "FirstScan",
                      Error => "ERR_ErrorData".ErrorLostPackage);
END_REGION

REGION Network 4: GlobalError
   RUNG wire#powerrail
      Contact( "ERR_ErrorData".ErrorEmergencyStop )
      wire#w1
      Coil( "MAN_LineModeData".Error )
   END_RUNG
   RUNG wire#powerrail
      Contact( "ERR_ErrorData".ErrorChangeMode )
   END_RUNG wire#w1
   RUNG wire#powerrail
      Contact( "ERR_ErrorData".ErrorLostPackage_B )
   END_RUNG wire#w1
   // the same network as SCL:
   "MAN_LineModeData".Error := "ERR_ErrorData".ErrorEmergencyStop OR "ERR_ErrorData".ErrorChangeMode OR "ERR_ErrorData".ErrorLostPackage_B;
END_REGION

REGION Network 5: ErrorLostPackage_B
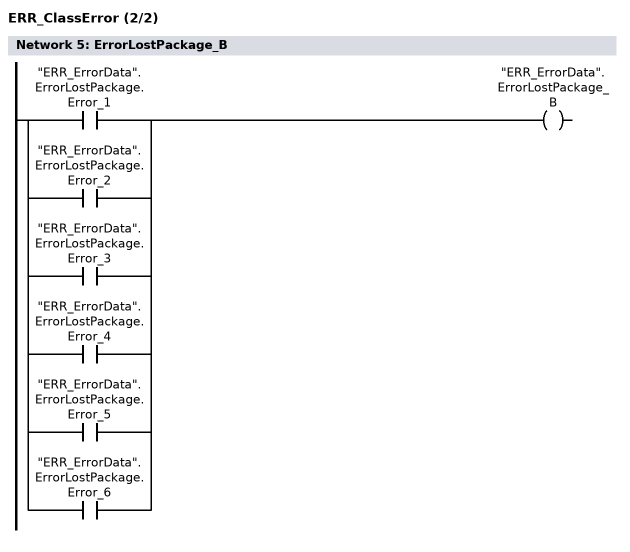
   RUNG wire#powerrail
      Contact( "ERR_ErrorData".ErrorLostPackage.Error_1 )
      wire#w1
      Coil( "ERR_ErrorData".ErrorLostPackage_B )
   END_RUNG
   RUNG wire#powerrail
      Contact( "ERR_ErrorData".ErrorLostPackage.Error_2 )
   END_RUNG wire#w1
   RUNG wire#powerrail
      Contact( "ERR_ErrorData".ErrorLostPackage.Error_3 )
   END_RUNG wire#w1
   RUNG wire#powerrail
      Contact( "ERR_ErrorData".ErrorLostPackage.Error_4 )
   END_RUNG wire#w1
   RUNG wire#powerrail
      Contact( "ERR_ErrorData".ErrorLostPackage.Error_5 )
   END_RUNG wire#w1
   RUNG wire#powerrail
      Contact( "ERR_ErrorData".ErrorLostPackage.Error_6 )
   END_RUNG wire#w1
   // the same network as SCL:
   "ERR_ErrorData".ErrorLostPackage_B := "ERR_ErrorData".ErrorLostPackage.Error_1 OR "ERR_ErrorData".ErrorLostPackage.Error_2 OR "ERR_ErrorData".ErrorLostPackage.Error_3 OR "ERR_ErrorData".ErrorLostPackage.Error_4 OR "ERR_ErrorData".ErrorLostPackage.Error_5 OR "ERR_ErrorData".ErrorLostPackage.Error_6;
END_REGION
END_FUNCTION

FUNCTION_BLOCK "ERR_EStop"   // FB6, LAD
{ S7_Optimized_Access := 'TRUE' }
VERSION : 0.1
// stored: AutoNumber true, IsIECCheckEnabled false, IsRetainMemResEnabled false, MemoryReserve 100, SetENOAutomatically false, UDAEnableTagReadback false
   VAR_INPUT
      EStopButton : Bool;
      ResetButton : Bool;
   END_VAR
   VAR_OUTPUT
      Error : Bool;
   END_VAR
   VAR
      P_ResetButton : Bool;
   END_VAR
   VAR_TEMP   // added for the SCL form of the ladder/FBD networks
      _w1 : Bool;
   END_VAR
BEGIN

REGION Network 1
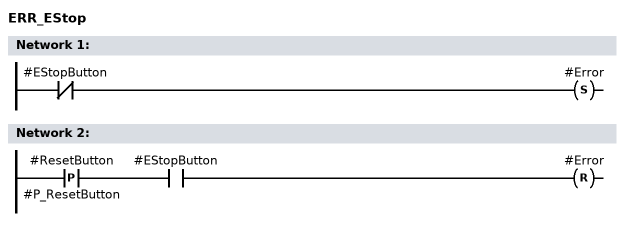
   RUNG wire#powerrail
      I_Contact( #EStopButton )
      S_Coil( #Error )
   END_RUNG
   // the same network as SCL:
   IF NOT #EStopButton THEN #Error := TRUE; END_IF;
END_REGION

REGION Network 2
   RUNG wire#powerrail
      P_Contact(operand := #ResetButton, bit := #P_ResetButton)
      Contact( #EStopButton )
      R_Coil( #Error )
   END_RUNG
   // the same network as SCL:
   #_w1 := #ResetButton AND NOT #P_ResetButton;   // rising edge of #ResetButton
   #P_ResetButton := #ResetButton;
   IF #_w1 AND #EStopButton THEN #Error := FALSE; END_IF;
END_REGION
END_FUNCTION_BLOCK

FUNCTION_BLOCK "ERR_ChangeMode"   // FB10, LAD
{ S7_Optimized_Access := 'TRUE' }
VERSION : 0.1
// stored: AutoNumber true, IsIECCheckEnabled false, IsRetainMemResEnabled false, MemoryReserve 100, SetENOAutomatically false, UDAEnableTagReadback false
   VAR_INPUT
      StartLine : Bool;
      StopLine : Bool;
      ModeAuto : Bool;
      ModeManual : Bool;
      ResetButton : Bool;
      AlarmSiren : Bool;
      FirstScan : Bool;
   END_VAR
   VAR_OUTPUT
      Error : Bool;
   END_VAR
   VAR
      S1 : Bool;
      S2 : Bool;
      S3 : Bool;
      S4 : Bool;
      S5 : Bool;
      P_ResetButton : Bool;
   END_VAR
   VAR_TEMP   // added for the SCL form of the ladder/FBD networks
      _w1 : Bool;
   END_VAR
BEGIN

REGION Network 1
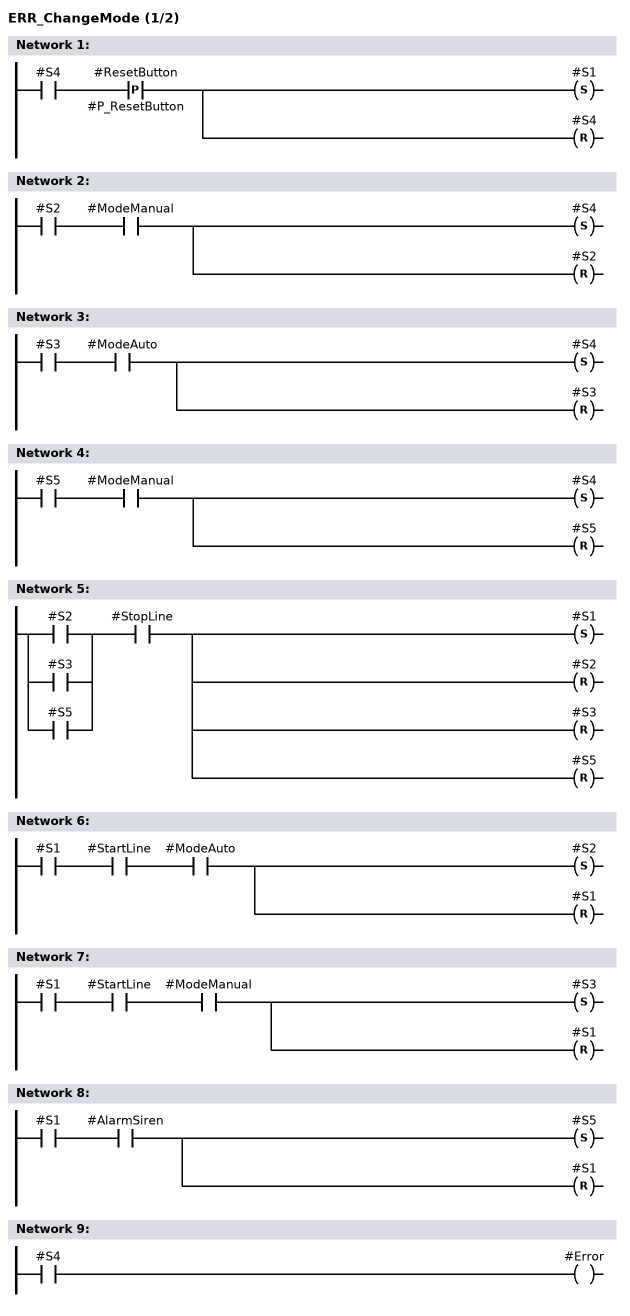
   RUNG wire#powerrail
      Contact( #S4 )
      P_Contact(operand := #ResetButton, bit := #P_ResetButton)
      wire#w1
      S_Coil( #S1 )
   END_RUNG
   RUNG wire#w1
      R_Coil( #S4 )
   END_RUNG
   // the same network as SCL:
   #_w1 := #S4 AND #ResetButton AND NOT #P_ResetButton;   // rising edge of #ResetButton
   #P_ResetButton := #ResetButton;
   IF #_w1 THEN
       #S1 := TRUE;
       #S4 := FALSE;
   END_IF;
END_REGION

REGION Network 2
   RUNG wire#powerrail
      Contact( #S2 )
      Contact( #ModeManual )
      wire#w1
      S_Coil( #S4 )
   END_RUNG
   RUNG wire#w1
      R_Coil( #S2 )
   END_RUNG
   // the same network as SCL:
   IF #S2 AND #ModeManual THEN
       #S4 := TRUE;
       #S2 := FALSE;
   END_IF;
END_REGION

REGION Network 3
   RUNG wire#powerrail
      Contact( #S3 )
      Contact( #ModeAuto )
      wire#w1
      S_Coil( #S4 )
   END_RUNG
   RUNG wire#w1
      R_Coil( #S3 )
   END_RUNG
   // the same network as SCL:
   IF #S3 AND #ModeAuto THEN
       #S4 := TRUE;
       #S3 := FALSE;
   END_IF;
END_REGION

REGION Network 4
   RUNG wire#powerrail
      Contact( #S5 )
      Contact( #ModeManual )
      wire#w1
      S_Coil( #S4 )
   END_RUNG
   RUNG wire#w1
      R_Coil( #S5 )
   END_RUNG
   // the same network as SCL:
   IF #S5 AND #ModeManual THEN
       #S4 := TRUE;
       #S5 := FALSE;
   END_IF;
END_REGION

REGION Network 5
   RUNG wire#powerrail
      Contact( #S2 )
      wire#w1
      Contact( #StopLine )
      wire#w2
      S_Coil( #S1 )
   END_RUNG
   RUNG wire#powerrail
      Contact( #S3 )
   END_RUNG wire#w1
   RUNG wire#powerrail
      Contact( #S5 )
   END_RUNG wire#w1
   RUNG wire#w2
      R_Coil( #S2 )
   END_RUNG
   RUNG wire#w2
      R_Coil( #S3 )
   END_RUNG
   RUNG wire#w2
      R_Coil( #S5 )
   END_RUNG
   // the same network as SCL:
   IF (#S2 OR #S3 OR #S5) AND #StopLine THEN #S1 := TRUE; END_IF;
   #_w1 := (#S2 OR #S3 OR #S5) AND #StopLine;
   IF #_w1 THEN
       #S2 := FALSE;
       #S3 := FALSE;
       #S5 := FALSE;
   END_IF;
END_REGION

REGION Network 6
   RUNG wire#powerrail
      Contact( #S1 )
      Contact( #StartLine )
      Contact( #ModeAuto )
      wire#w1
      S_Coil( #S2 )
   END_RUNG
   RUNG wire#w1
      R_Coil( #S1 )
   END_RUNG
   // the same network as SCL:
   IF #S1 AND #StartLine AND #ModeAuto THEN
       #S2 := TRUE;
       #S1 := FALSE;
   END_IF;
END_REGION

REGION Network 7
   RUNG wire#powerrail
      Contact( #S1 )
      Contact( #StartLine )
      Contact( #ModeManual )
      wire#w1
      S_Coil( #S3 )
   END_RUNG
   RUNG wire#w1
      R_Coil( #S1 )
   END_RUNG
   // the same network as SCL:
   IF #S1 AND #StartLine AND #ModeManual THEN
       #S3 := TRUE;
       #S1 := FALSE;
   END_IF;
END_REGION

REGION Network 8
   RUNG wire#powerrail
      Contact( #S1 )
      Contact( #AlarmSiren )
      wire#w1
      S_Coil( #S5 )
   END_RUNG
   RUNG wire#w1
      R_Coil( #S1 )
   END_RUNG
   // the same network as SCL:
   IF #S1 AND #AlarmSiren THEN
       #S5 := TRUE;
       #S1 := FALSE;
   END_IF;
END_REGION

REGION Network 9
   RUNG wire#powerrail
      Contact( #S4 )
      Coil( #Error )
   END_RUNG
   // the same network as SCL:
   #Error := #S4;
END_REGION

REGION Network 10
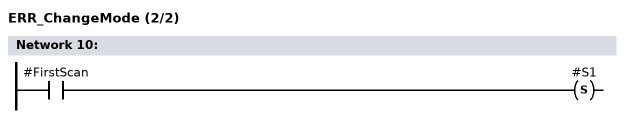
   RUNG wire#powerrail
      Contact( #FirstScan )
      S_Coil( #S1 )
   END_RUNG
   // the same network as SCL:
   IF #FirstScan THEN #S1 := TRUE; END_IF;
END_REGION
END_FUNCTION_BLOCK

FUNCTION "ERR_LostPackages" : Void   // FC12, LAD
{ S7_Optimized_Access := 'TRUE' }
VERSION : 0.1
// stored: AutoNumber true, IsIECCheckEnabled false, SetENOAutomatically false, UDAEnableTagReadback false
   VAR_INPUT
      StartLine : Bool;
      StopLine : Bool;
      AutoMode : Bool;
      ResetButton : Bool;
      FirstScan : Bool;
   END_VAR
   VAR_OUTPUT
      Error : "stt_LostPackageError";
   END_VAR
BEGIN

REGION Network 1: Call: LostPackage - error 1
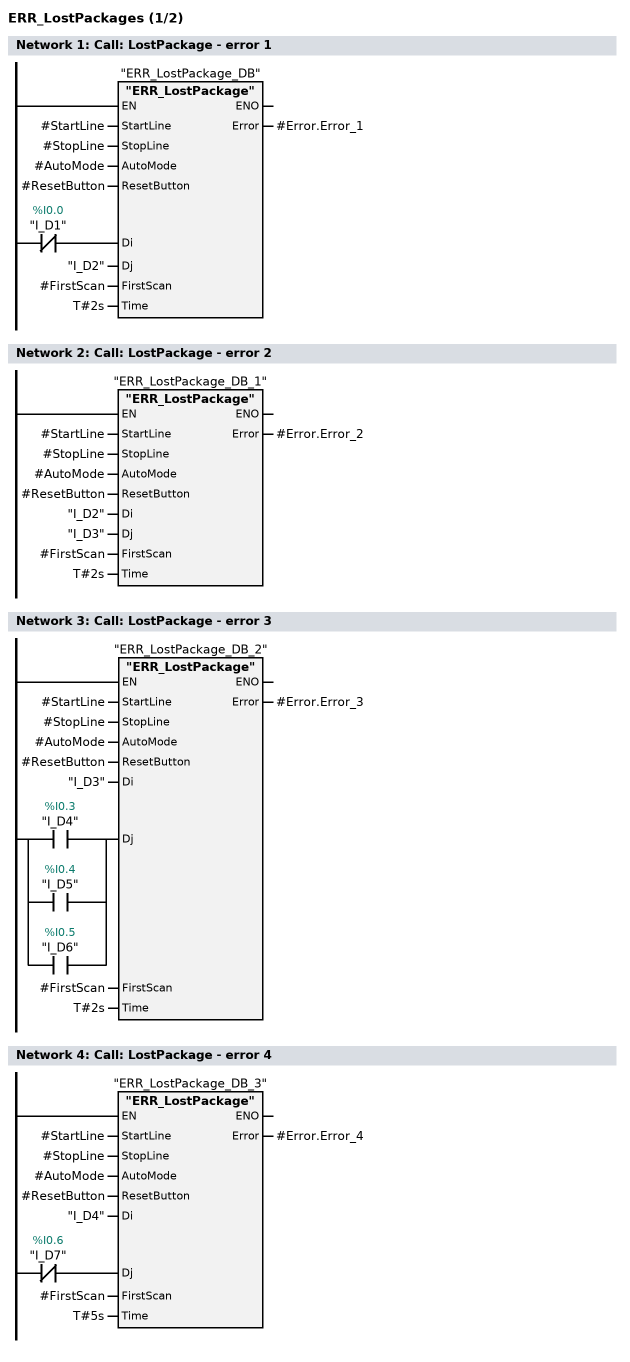
   RUNG wire#powerrail
      "ERR_LostPackage_DB"(Di := wire#w1, StartLine := #StartLine, StopLine := #StopLine, AutoMode := #AutoMode, ResetButton := #ResetButton, Dj := "I_D2", FirstScan := #FirstScan, "Time" := T#2s, Error => #Error.Error_1)
   END_RUNG
   RUNG wire#powerrail
      I_Contact( "I_D1" )
   END_RUNG wire#w1
   // the same network as SCL:
   "ERR_LostPackage_DB"(StartLine := #StartLine,   // "ERR_LostPackage"
                        StopLine := #StopLine,
                        AutoMode := #AutoMode,
                        ResetButton := #ResetButton,
                        Di := NOT "I_D1",
                        Dj := "I_D2",
                        FirstScan := #FirstScan,
                        "Time" := T#2s,
                        Error => #Error.Error_1);
END_REGION

REGION Network 2: Call: LostPackage - error 2
   RUNG wire#powerrail
      "ERR_LostPackage_DB_1"(StartLine := #StartLine, StopLine := #StopLine, AutoMode := #AutoMode, ResetButton := #ResetButton, Di := "I_D2", Dj := "I_D3", FirstScan := #FirstScan, "Time" := T#2s, Error => #Error.Error_2)
   END_RUNG
   // the same network as SCL:
   "ERR_LostPackage_DB_1"(StartLine := #StartLine,   // "ERR_LostPackage"
                          StopLine := #StopLine,
                          AutoMode := #AutoMode,
                          ResetButton := #ResetButton,
                          Di := "I_D2",
                          Dj := "I_D3",
                          FirstScan := #FirstScan,
                          "Time" := T#2s,
                          Error => #Error.Error_2);
END_REGION

REGION Network 3: Call: LostPackage - error 3
   RUNG wire#powerrail
      "ERR_LostPackage_DB_2"(Dj := wire#w1, StartLine := #StartLine, StopLine := #StopLine, AutoMode := #AutoMode, ResetButton := #ResetButton, Di := "I_D3", FirstScan := #FirstScan, "Time" := T#2s, Error => #Error.Error_3)
   END_RUNG
   RUNG wire#powerrail
      Contact( "I_D4" )
   END_RUNG wire#w1
   RUNG wire#powerrail
      Contact( "I_D5" )
   END_RUNG wire#w1
   RUNG wire#powerrail
      Contact( "I_D6" )
   END_RUNG wire#w1
   // the same network as SCL:
   "ERR_LostPackage_DB_2"(StartLine := #StartLine,   // "ERR_LostPackage"
                          StopLine := #StopLine,
                          AutoMode := #AutoMode,
                          ResetButton := #ResetButton,
                          Di := "I_D3",
                          Dj := "I_D4" OR "I_D5" OR "I_D6",
                          FirstScan := #FirstScan,
                          "Time" := T#2s,
                          Error => #Error.Error_3);
END_REGION

REGION Network 4: Call: LostPackage - error 4
   RUNG wire#powerrail
      "ERR_LostPackage_DB_3"(Dj := wire#w1, StartLine := #StartLine, StopLine := #StopLine, AutoMode := #AutoMode, ResetButton := #ResetButton, Di := "I_D4", FirstScan := #FirstScan, "Time" := T#5s, Error => #Error.Error_4)
   END_RUNG
   RUNG wire#powerrail
      I_Contact( "I_D7" )
   END_RUNG wire#w1
   // the same network as SCL:
   "ERR_LostPackage_DB_3"(StartLine := #StartLine,   // "ERR_LostPackage"
                          StopLine := #StopLine,
                          AutoMode := #AutoMode,
                          ResetButton := #ResetButton,
                          Di := "I_D4",
                          Dj := NOT "I_D7",
                          FirstScan := #FirstScan,
                          "Time" := T#5s,
                          Error => #Error.Error_4);
END_REGION

REGION Network 5: Call: LostPackage - error 5
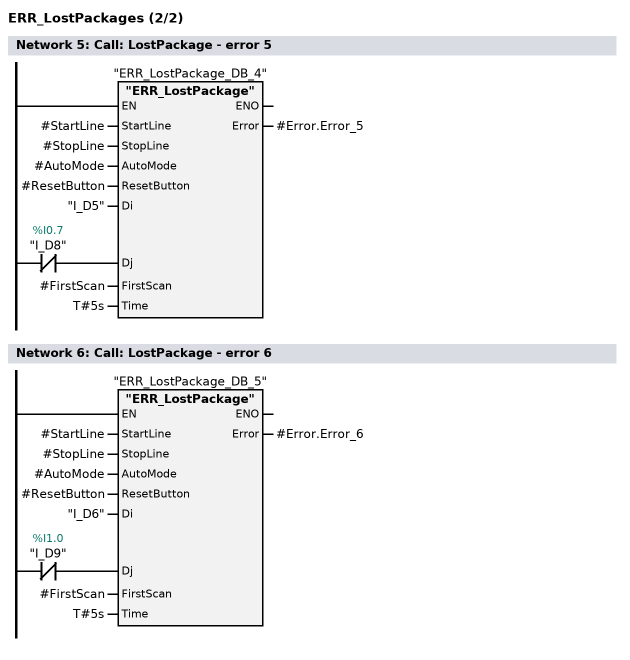
   RUNG wire#powerrail
      "ERR_LostPackage_DB_4"(Dj := wire#w1, StartLine := #StartLine, StopLine := #StopLine, AutoMode := #AutoMode, ResetButton := #ResetButton, Di := "I_D5", FirstScan := #FirstScan, "Time" := T#5s, Error => #Error.Error_5)
   END_RUNG
   RUNG wire#powerrail
      I_Contact( "I_D8" )
   END_RUNG wire#w1
   // the same network as SCL:
   "ERR_LostPackage_DB_4"(StartLine := #StartLine,   // "ERR_LostPackage"
                          StopLine := #StopLine,
                          AutoMode := #AutoMode,
                          ResetButton := #ResetButton,
                          Di := "I_D5",
                          Dj := NOT "I_D8",
                          FirstScan := #FirstScan,
                          "Time" := T#5s,
                          Error => #Error.Error_5);
END_REGION

REGION Network 6: Call: LostPackage - error 6
   RUNG wire#powerrail
      "ERR_LostPackage_DB_5"(Dj := wire#w1, StartLine := #StartLine, StopLine := #StopLine, AutoMode := #AutoMode, ResetButton := #ResetButton, Di := "I_D6", FirstScan := #FirstScan, "Time" := T#5s, Error => #Error.Error_6)
   END_RUNG
   RUNG wire#powerrail
      I_Contact( "I_D9" )
   END_RUNG wire#w1
   // the same network as SCL:
   "ERR_LostPackage_DB_5"(StartLine := #StartLine,   // "ERR_LostPackage"
                          StopLine := #StopLine,
                          AutoMode := #AutoMode,
                          ResetButton := #ResetButton,
                          Di := "I_D6",
                          Dj := NOT "I_D9",
                          FirstScan := #FirstScan,
                          "Time" := T#5s,
                          Error => #Error.Error_6);
END_REGION
END_FUNCTION

FUNCTION_BLOCK "ERR_LostPackage"   // FB12, LAD
TITLE = Lost Package - Sequential algorithm
{ S7_Optimized_Access := 'TRUE' }
VERSION : 0.1
// stored: AutoNumber true, IsIECCheckEnabled false, IsRetainMemResEnabled false, MemoryReserve 100, SetENOAutomatically false, UDAEnableTagReadback false
   VAR_INPUT
      StartLine : Bool;
      StopLine : Bool;
      AutoMode : Bool;
      ResetButton : Bool;
      Di : Bool;
      Dj : Bool;
      FirstScan : Bool;
      "Time" : Time;
   END_VAR
   VAR_OUTPUT
      Error : Bool;
   END_VAR
   VAR
      S1 : Bool;
      S2 : Bool;
      S3 : Bool;
      t1 : Bool;
      P_ResetButton : Bool;
      IEC_Timer_0_Instance { ExternalAccessible := 'False'; ExternalVisible := 'False'; ExternalWritable := 'False'} : TON_TIME;
   END_VAR
   VAR_TEMP   // added for the SCL form of the ladder/FBD networks
      _w1 : Bool;
   END_VAR
BEGIN

REGION Network 1: Step 3-1
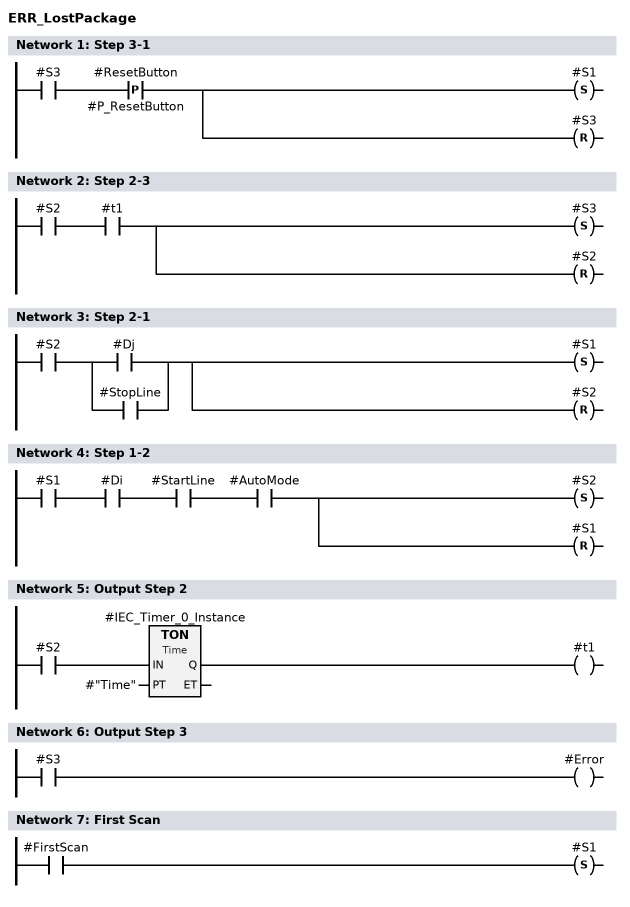
   RUNG wire#powerrail
      Contact( #S3 )
      P_Contact(operand := #ResetButton, bit := #P_ResetButton)
      wire#w1
      S_Coil( #S1 )
   END_RUNG
   RUNG wire#w1
      R_Coil( #S3 )
   END_RUNG
   // the same network as SCL:
   #_w1 := #S3 AND #ResetButton AND NOT #P_ResetButton;   // rising edge of #ResetButton
   #P_ResetButton := #ResetButton;
   IF #_w1 THEN
       #S1 := TRUE;
       #S3 := FALSE;
   END_IF;
END_REGION

REGION Network 2: Step 2-3
   RUNG wire#powerrail
      Contact( #S2 )
      Contact( #t1 )
      wire#w1
      S_Coil( #S3 )
   END_RUNG
   RUNG wire#w1
      R_Coil( #S2 )
   END_RUNG
   // the same network as SCL:
   IF #S2 AND #t1 THEN
       #S3 := TRUE;
       #S2 := FALSE;
   END_IF;
END_REGION

REGION Network 3: Step 2-1
   RUNG wire#powerrail
      Contact( #S2 )
      wire#w1
      Contact( #Dj )
      wire#w2
      S_Coil( #S1 )
   END_RUNG
   RUNG wire#w1
      Contact( #StopLine )
   END_RUNG wire#w2
   RUNG wire#w2
      R_Coil( #S2 )
   END_RUNG
   // the same network as SCL:
   IF #S2 AND (#Dj OR #StopLine) THEN
       #S1 := TRUE;
       #S2 := FALSE;
   END_IF;
END_REGION

REGION Network 4: Step 1-2
   RUNG wire#powerrail
      Contact( #S1 )
      Contact( #Di )
      Contact( #StartLine )
      Contact( #AutoMode )
      wire#w1
      S_Coil( #S2 )
   END_RUNG
   RUNG wire#w1
      R_Coil( #S1 )
   END_RUNG
   // the same network as SCL:
   IF #S1 AND #Di AND #StartLine AND #AutoMode THEN
       #S2 := TRUE;
       #S1 := FALSE;
   END_IF;
END_REGION

REGION Network 5: Output Step 2
   RUNG wire#powerrail
      Contact( #S2 )
      { S7_Templates := "time_type := Time" } #IEC_Timer_0_Instance.TON(pt := #"Time", et =>)
      Coil( #t1 )
   END_RUNG
   // the same network as SCL:
   #IEC_Timer_0_Instance(IN := #S2, PT := #"Time");   // TON
   #t1 := #IEC_Timer_0_Instance.Q;
END_REGION

REGION Network 6: Output Step 3
   RUNG wire#powerrail
      Contact( #S3 )
      Coil( #Error )
   END_RUNG
   // the same network as SCL:
   #Error := #S3;
END_REGION

REGION Network 7: First Scan
   RUNG wire#powerrail
      Contact( #FirstScan )
      S_Coil( #S1 )
   END_RUNG
   // the same network as SCL:
   IF #FirstScan THEN #S1 := TRUE; END_IF;
END_REGION
END_FUNCTION_BLOCK

ORGANIZATION_BLOCK "Startup"   // OB100, LAD, Startup
TITLE = "Complete Restart"
{ S7_Optimized_Access := 'TRUE' }
VERSION : 0.1
// stored: AutoNumber true, IsIECCheckEnabled false, SetENOAutomatically false
   VAR_INPUT
      LostRetentive : Bool;   // True if retentive data are lost
      LostRTC : Bool;   // True if date and time are lost
   END_VAR
BEGIN
END_ORGANIZATION_BLOCK

ORGANIZATION_BLOCK "HW_Weight"   // OB30, LAD, CyclicInterrupt
{ S7_Optimized_Access := 'TRUE' }
VERSION : 0.1
// stored: AutoNumber true, IsIECCheckEnabled false, SetENOAutomatically false
   VAR_INPUT
      Initial_Call : Bool;   // Initial call of this OB
      Event_Count : Int;   // Events discarded
   END_VAR
   VAR_TEMP
      Work : Bool;
   END_VAR
   VAR_TEMP   // added for the SCL form of the ladder/FBD networks
      _w1 : Bool;
   END_VAR
BEGIN

REGION Network 1: Call: MovingAverageFilter
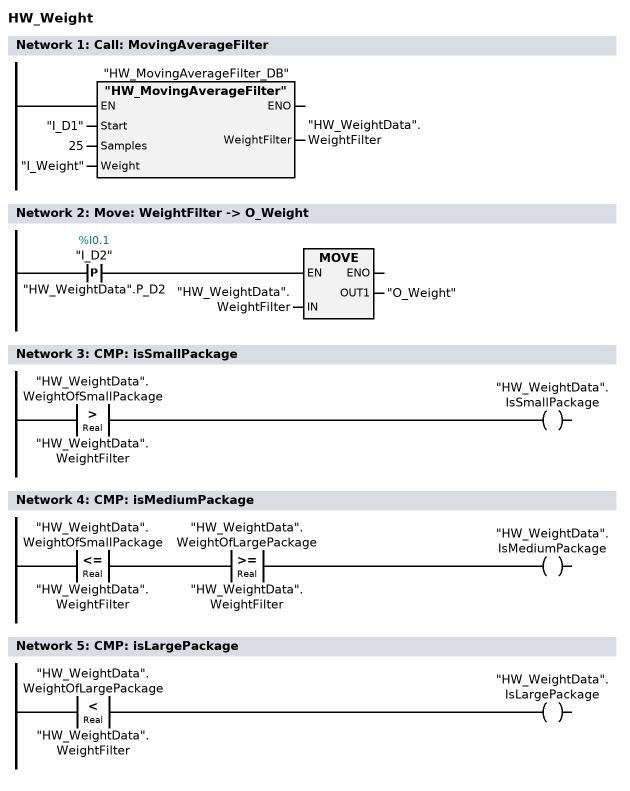
   RUNG wire#powerrail
      "HW_MovingAverageFilter_DB"(Start := "I_D1", Samples := 25, Weight := "I_Weight", WeightFilter => "HW_WeightData".WeightFilter)
   END_RUNG
   // the same network as SCL:
   "HW_MovingAverageFilter_DB"(Start := "I_D1",   // "HW_MovingAverageFilter"
                           Samples := 25,
                           Weight := "I_Weight",
                           WeightFilter => "HW_WeightData".WeightFilter);
END_REGION

REGION Network 2: Move: WeightFilter -> O_Weight
   RUNG wire#powerrail
      P_Contact(operand := "I_D2", bit := "HW_WeightData".P_D2)
      Move(in := "HW_WeightData".WeightFilter, out1 => "O_Weight")
   END_RUNG
   // the same network as SCL:
   #_w1 := "I_D2" AND NOT "HW_WeightData".P_D2;   // rising edge of "I_D2"
   "HW_WeightData".P_D2 := "I_D2";
   IF #_w1 THEN "O_Weight" := "HW_WeightData".WeightFilter; END_IF;
END_REGION

REGION Network 3: CMP: isSmallPackage
   RUNG wire#powerrail
      { S7_Templates := "SrcType := Real" } GT_Contact(in1 := "HW_WeightData".WeightOfSmallPackage, in2 := "HW_WeightData".WeightFilter)
      Coil( "HW_WeightData".IsSmallPackage )
   END_RUNG
   // the same network as SCL:
   "HW_WeightData".IsSmallPackage := "HW_WeightData".WeightOfSmallPackage > "HW_WeightData".WeightFilter;
END_REGION

REGION Network 4: CMP: isMediumPackage
   RUNG wire#powerrail
      { S7_Templates := "SrcType := Real" } LE_Contact(in1 := "HW_WeightData".WeightOfSmallPackage, in2 := "HW_WeightData".WeightFilter)
      { S7_Templates := "SrcType := Real" } GE_Contact(in1 := "HW_WeightData".WeightOfLargePackage, in2 := "HW_WeightData".WeightFilter)
      Coil( "HW_WeightData".IsMediumPackage )
   END_RUNG
   // the same network as SCL:
   "HW_WeightData".IsMediumPackage := ("HW_WeightData".WeightOfSmallPackage <= "HW_WeightData".WeightFilter) AND ("HW_WeightData".WeightOfLargePackage >= "HW_WeightData".WeightFilter);
END_REGION

REGION Network 5: CMP: isLargePackage
   RUNG wire#powerrail
      { S7_Templates := "SrcType := Real" } LT_Contact(in1 := "HW_WeightData".WeightOfLargePackage, in2 := "HW_WeightData".WeightFilter)
      Coil( "HW_WeightData".IsLargePackage )
   END_RUNG
   // the same network as SCL:
   "HW_WeightData".IsLargePackage := "HW_WeightData".WeightOfLargePackage < "HW_WeightData".WeightFilter;
END_REGION
END_ORGANIZATION_BLOCK

FUNCTION_BLOCK "HW_MovingAverageFilter"
{ S7_Optimized_Access := 'TRUE' }
VERSION : 0.1
   VAR_INPUT 
      Start : Bool;
      Samples : Int;
      Weight : Real;
   END_VAR

   VAR_OUTPUT 
      WeightFilter : Real;
   END_VAR

   VAR 
      Bufor : Array[0..99] of Real;
   END_VAR

   VAR_TEMP 
      Sum : Real;
      index : Int;
   END_VAR


BEGIN
	IF #Start THEN
	    FOR #index := (#Samples - 2) TO 0 BY -1 DO
	        #Bufor[#index + 1] := #Bufor[#index];
	    END_FOR;
	    
	    #Bufor[0] := #Weight;
	    #Sum := 0;
	    
	    FOR #index := 0 TO (#Samples - 1) DO
	        #Sum := #Sum + #Bufor[#index];
	    END_FOR;
	    
	    #WeightFilter := #Sum / #Samples;
	ELSE
	    #WeightFilter := 0;
	END_IF;
	
	
	
	
	
	
	
	
	
END_FUNCTION_BLOCK

FUNCTION "MAN_ClassManagement" : Void   // FC3, LAD
{ S7_Optimized_Access := 'TRUE' }
VERSION : 0.1
// stored: AutoNumber true, IsIECCheckEnabled false, SetENOAutomatically false, UDAEnableTagReadback false
BEGIN

REGION Network 1: Call: ChooseMode
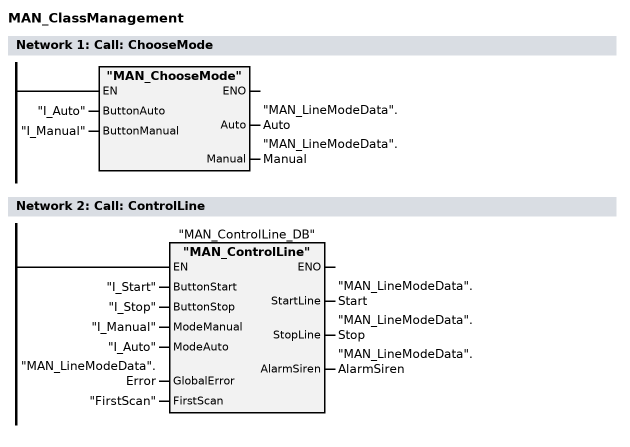
   RUNG wire#powerrail
      "MAN_ChooseMode"(ButtonAuto := "I_Auto", ButtonManual := "I_Manual", Auto => "MAN_LineModeData".Auto, Manual => "MAN_LineModeData".Manual)
   END_RUNG
   // the same network as SCL:
   "MAN_ChooseMode"(ButtonAuto := "I_Auto",
                    ButtonManual := "I_Manual",
                    Auto => "MAN_LineModeData".Auto,
                    Manual => "MAN_LineModeData".Manual);
END_REGION

REGION Network 2: Call: ControlLine
   RUNG wire#powerrail
      "MAN_ControlLine_DB"(ButtonStart := "I_Start", ButtonStop := "I_Stop", ModeManual := "I_Manual", ModeAuto := "I_Auto", GlobalError := "MAN_LineModeData".Error, FirstScan := "FirstScan", StartLine => "MAN_LineModeData".Start, StopLine => "MAN_LineModeData".Stop, AlarmSiren => "MAN_LineModeData".AlarmSiren)
   END_RUNG
   // the same network as SCL:
   "MAN_ControlLine_DB"(ButtonStart := "I_Start",   // "MAN_ControlLine"
                        ButtonStop := "I_Stop",
                        ModeManual := "I_Manual",
                        ModeAuto := "I_Auto",
                        GlobalError := "MAN_LineModeData".Error,
                        FirstScan := "FirstScan",
                        StartLine => "MAN_LineModeData".Start,
                        StopLine => "MAN_LineModeData".Stop,
                        AlarmSiren => "MAN_LineModeData".AlarmSiren);
END_REGION
END_FUNCTION

FUNCTION "HW_ClassHardware" : Void   // FC5, LAD
{ S7_Optimized_Access := 'TRUE' }
VERSION : 0.1
// stored: AutoNumber true, IsIECCheckEnabled false, SetENOAutomatically false, UDAEnableTagReadback false
BEGIN
END_FUNCTION

FUNCTION_BLOCK "HW_MotorControle"   // FB1, LAD
{ S7_Optimized_Access := 'TRUE' }
VERSION : 0.1
// stored: AutoNumber true, IsIECCheckEnabled false, IsRetainMemResEnabled false, MemoryReserve 100, SetENOAutomatically false, UDAEnableTagReadback false
   VAR_INPUT
      inConveyor : "stt_Motor";
      FirstScan : Bool;
   END_VAR
   VAR_OUTPUT
      Conveyor : Real;
   END_VAR
   VAR
      S1 : Bool;
      S2 : Bool;
      S3 : Bool;
      S4 : Bool;
      S5 : Bool;
      t1 : Bool;
      t2 : Bool;
      speedLeft : Real;
      IEC_Timer_0_Instance { ExternalAccessible := 'False'; ExternalVisible := 'False'; ExternalWritable := 'False'} : TON_TIME;
      IEC_Timer_0_Instance_1 { ExternalAccessible := 'False'; ExternalVisible := 'False'; ExternalWritable := 'False'} : TON_TIME;
   END_VAR
BEGIN

REGION Network 1: Step 2-1
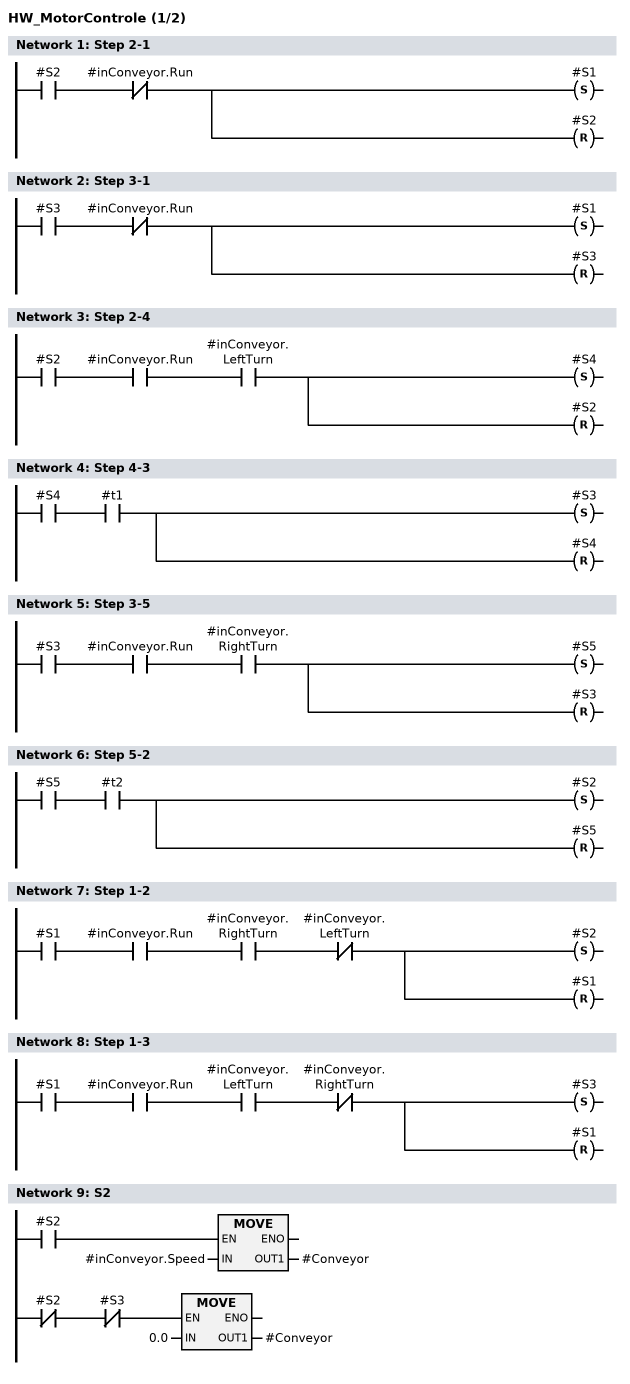
   RUNG wire#powerrail
      Contact( #S2 )
      I_Contact( #inConveyor.Run )
      wire#w1
      S_Coil( #S1 )
   END_RUNG
   RUNG wire#w1
      R_Coil( #S2 )
   END_RUNG
   // the same network as SCL:
   IF #S2 AND NOT #inConveyor.Run THEN
       #S1 := TRUE;
       #S2 := FALSE;
   END_IF;
END_REGION

REGION Network 2: Step 3-1
   RUNG wire#powerrail
      Contact( #S3 )
      I_Contact( #inConveyor.Run )
      wire#w1
      S_Coil( #S1 )
   END_RUNG
   RUNG wire#w1
      R_Coil( #S3 )
   END_RUNG
   // the same network as SCL:
   IF #S3 AND NOT #inConveyor.Run THEN
       #S1 := TRUE;
       #S3 := FALSE;
   END_IF;
END_REGION

REGION Network 3: Step 2-4
   RUNG wire#powerrail
      Contact( #S2 )
      Contact( #inConveyor.Run )
      Contact( #inConveyor.LeftTurn )
      wire#w1
      S_Coil( #S4 )
   END_RUNG
   RUNG wire#w1
      R_Coil( #S2 )
   END_RUNG
   // the same network as SCL:
   IF #S2 AND #inConveyor.Run AND #inConveyor.LeftTurn THEN
       #S4 := TRUE;
       #S2 := FALSE;
   END_IF;
END_REGION

REGION Network 4: Step 4-3
   RUNG wire#powerrail
      Contact( #S4 )
      Contact( #t1 )
      wire#w1
      S_Coil( #S3 )
   END_RUNG
   RUNG wire#w1
      R_Coil( #S4 )
   END_RUNG
   // the same network as SCL:
   IF #S4 AND #t1 THEN
       #S3 := TRUE;
       #S4 := FALSE;
   END_IF;
END_REGION

REGION Network 5: Step 3-5
   RUNG wire#powerrail
      Contact( #S3 )
      Contact( #inConveyor.Run )
      Contact( #inConveyor.RightTurn )
      wire#w1
      S_Coil( #S5 )
   END_RUNG
   RUNG wire#w1
      R_Coil( #S3 )
   END_RUNG
   // the same network as SCL:
   IF #S3 AND #inConveyor.Run AND #inConveyor.RightTurn THEN
       #S5 := TRUE;
       #S3 := FALSE;
   END_IF;
END_REGION

REGION Network 6: Step 5-2
   RUNG wire#powerrail
      Contact( #S5 )
      Contact( #t2 )
      wire#w1
      S_Coil( #S2 )
   END_RUNG
   RUNG wire#w1
      R_Coil( #S5 )
   END_RUNG
   // the same network as SCL:
   IF #S5 AND #t2 THEN
       #S2 := TRUE;
       #S5 := FALSE;
   END_IF;
END_REGION

REGION Network 7: Step 1-2
   RUNG wire#powerrail
      Contact( #S1 )
      Contact( #inConveyor.Run )
      Contact( #inConveyor.RightTurn )
      I_Contact( #inConveyor.LeftTurn )
      wire#w1
      S_Coil( #S2 )
   END_RUNG
   RUNG wire#w1
      R_Coil( #S1 )
   END_RUNG
   // the same network as SCL:
   IF #S1 AND #inConveyor.Run AND #inConveyor.RightTurn AND NOT #inConveyor.LeftTurn THEN
       #S2 := TRUE;
       #S1 := FALSE;
   END_IF;
END_REGION

REGION Network 8: Step 1-3
   RUNG wire#powerrail
      Contact( #S1 )
      Contact( #inConveyor.Run )
      Contact( #inConveyor.LeftTurn )
      I_Contact( #inConveyor.RightTurn )
      wire#w1
      S_Coil( #S3 )
   END_RUNG
   RUNG wire#w1
      R_Coil( #S1 )
   END_RUNG
   // the same network as SCL:
   IF #S1 AND #inConveyor.Run AND #inConveyor.LeftTurn AND NOT #inConveyor.RightTurn THEN
       #S3 := TRUE;
       #S1 := FALSE;
   END_IF;
END_REGION

REGION Network 9: S2
   RUNG wire#powerrail
      Contact( #S2 )
      Move(in := #inConveyor.Speed, out1 => #Conveyor)
   END_RUNG
   RUNG wire#powerrail
      I_Contact( #S2 )
      I_Contact( #S3 )
      Move(in := 0.0, out1 => #Conveyor)
   END_RUNG
   // the same network as SCL:
   IF #S2 THEN #Conveyor := #inConveyor.Speed; END_IF;
   IF NOT #S2 AND NOT #S3 THEN #Conveyor := 0.0; END_IF;
END_REGION

REGION Network 10: S3
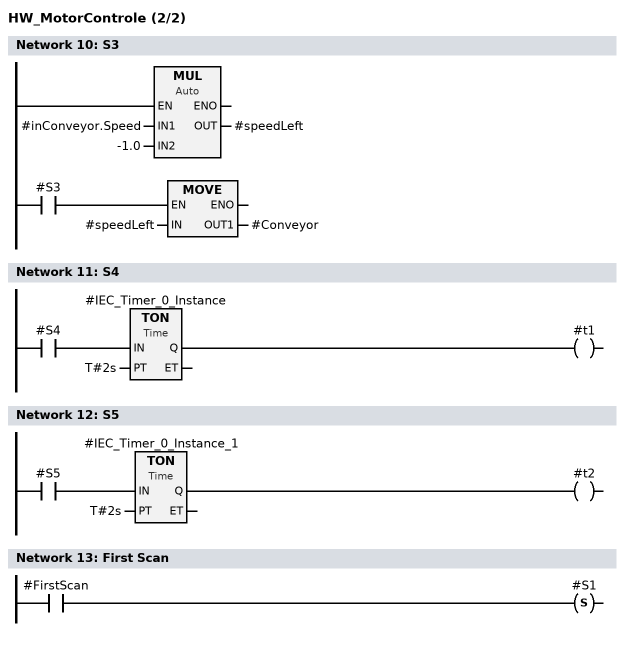
   RUNG wire#powerrail
      Mul(in1 := #inConveyor.Speed, in2 := -1.0, out => #speedLeft)
   END_RUNG
   RUNG wire#powerrail
      Contact( #S3 )
      Move(in := #speedLeft, out1 => #Conveyor)
   END_RUNG
   // the same network as SCL:
   #speedLeft := #inConveyor.Speed * (-1.0);
   IF #S3 THEN #Conveyor := #speedLeft; END_IF;
END_REGION

REGION Network 11: S4
   RUNG wire#powerrail
      Contact( #S4 )
      { S7_Templates := "time_type := Time" } #IEC_Timer_0_Instance.TON(pt := T#2s, et =>)
      Coil( #t1 )
   END_RUNG
   // the same network as SCL:
   #IEC_Timer_0_Instance(IN := #S4, PT := T#2s);   // TON
   #t1 := #IEC_Timer_0_Instance.Q;
END_REGION

REGION Network 12: S5
   RUNG wire#powerrail
      Contact( #S5 )
      { S7_Templates := "time_type := Time" } #IEC_Timer_0_Instance_1.TON(pt := T#2s, et =>)
      Coil( #t2 )
   END_RUNG
   // the same network as SCL:
   #IEC_Timer_0_Instance_1(IN := #S5, PT := T#2s);   // TON
   #t2 := #IEC_Timer_0_Instance_1.Q;
END_REGION

REGION Network 13: First Scan
   RUNG wire#powerrail
      Contact( #FirstScan )
      S_Coil( #S1 )
   END_RUNG
   // the same network as SCL:
   IF #FirstScan THEN #S1 := TRUE; END_IF;
END_REGION
END_FUNCTION_BLOCK

FUNCTION "H_ClassHMI" : Void   // FC6, LAD
{ S7_Optimized_Access := 'TRUE' }
VERSION : 0.1
// stored: AutoNumber true, IsIECCheckEnabled false, SetENOAutomatically false, UDAEnableTagReadback false
BEGIN
END_FUNCTION

FUNCTION "LOG_ButtonsLight" : Void   // FC14, LAD
{ S7_Optimized_Access := 'TRUE' }
VERSION : 0.1
// stored: AutoNumber true, IsIECCheckEnabled false, SetENOAutomatically false, UDAEnableTagReadback false
BEGIN

REGION Network 1: Button Start
